LIN {X 0,Y 573.448,Z 568.908,A -85,B 0,C 180,E1 -2263.285,E2 -2263.285} C_VEL
LIN {X 0,Y 573.59,Z 558.034,A -85,B 0,C 180,E1 -2264.544,E2 -2264.544} C_VEL
LIN {X 0,Y 573.831,Z 547.069,A -85,B 0,C 180,E1 -2265.631,E2 -2265.631} C_VEL
LIN {X 0,Y 574.091,Z 533.22,A -85,B 0,C 180,E1 -2266.811,E2 -2266.811} C_VEL
LIN {X 0,Y 574.357,Z 519.267,A -85,B 0,C 180,E1 -2267.813,E2 -2267.813} C_VEL
LIN {X 0,Y 574.661,Z 505.713,A -85,B 0,C 180,E1 -2268.633,E2 -2268.633} C_VEL
LIN {X 0,Y 574.868,Z 491.148,A -85,B 0,C 180,E1 -2269.364,E2 -2269.364} C_VEL
LIN {X 0,Y 575.123,Z 475.242,A -85,B 0,C 180,E1 -2270.008,E2 -2270.008} C_VEL
LIN {X 0,Y 575.358,Z 459.013,A -85,B 0,C 180,E1 -2270.513,E2 -2270.513} C_VEL
LIN {X 0,Y 575.478,Z 442.433,A -85,B 0,C 180,E1 -2270.882,E2 -2270.882} C_VEL
LIN {X 0,Y 576.09,Z 283.124,A -85,B 0,C 180,E1 -2272.978,E2 -2272.978} C_VEL
LIN {X 0,Y 576.127,Z 240.798,A -85,B 0,C 180,E1 -2273.539,E2 -2273.539} C_VEL
LIN {X 0,Y 575.049,Z 234.756,A -85,B 0,C 180,E1 -2273.688,E2 -2273.688} C_VEL
LIN {X 0,Y 575.522,Z 200.414,A -85,B 0,C 180,E1 -2276.665,E2 -2276.665} C_VEL
LIN {X 0,Y 575.558,Z 194.845,A -85,B 0,C 180,E1 -2277.153,E2 -2277.153} C_VEL
LIN {X 0,Y 573.24,Z 186.394,A -85,B 0,C 180,E1 -2278.027,E2 -2278.027} C_VEL
LIN {X 0,Y 573.215,Z 186.397,A -85,B 0,C 180,E1 -2280.994,E2 -2280.994} C_VEL
LIN {X 0,Y 573.261,Z 186.39,A -85,B 0,C 180,E1 -2283.524,E2 -2283.524} C_VEL
LIN {X 0,Y 573.19,Z 186.394,A -85,B 0,C 180,E1 -2286.053,E2 -2286.053} C_VEL
LIN {X 0,Y 573.239,Z 186.391,A -85,B 0,C 180,E1 -2288.702,E2 -2288.702} C_VEL
LIN {X 0,Y 573.211,Z 186.393,A -85,B 0,C 180,E1 -2291.591,E2 -2291.591} C_VEL
LIN {X 0,Y 573.221,Z 186.39,A -85,B 0,C 180,E1 -2294.334,E2 -2294.334} C_VEL
LIN {X 0,Y 573.234,Z 186.392,A -85,B 0,C 180,E1 -2297.359,E2 -2297.359} C_VEL
LIN {X 0,Y 573.233,Z 186.389,A -85,B 0,C 180,E1 -2300.392,E2 -2300.392} C_VEL
LIN {X 0,Y 573.249,Z 186.391,A -85,B 0,C 180,E1 -2303.077,E2 -2303.077} C_VEL
LIN {X 0,Y 573.258,Z 186.385,A -85,B 0,C 180,E1 -2305.671,E2 -2305.671} C_VEL
LIN {X 0,Y 573.242,Z 186.386,A -85,B 0,C 180,E1 -2308.185,E2 -2308.185} C_VEL
LIN {X 0,Y 573.254,Z 186.392,A -85,B 0,C 180,E1 -2310.634,E2 -2310.634} C_VEL
LIN {X 0,Y 573.246,Z 186.388,A -85,B 0,C 180,E1 -2313.024,E2 -2313.024} C_VEL
LIN {X 0,Y 573.269,Z 186.383,A -85,B 0,C 180,E1 -2315.366,E2 -2315.366} C_VEL
LIN {X 0,Y 573.224,Z 186.395,A -85,B 0,C 180,E1 -2318.419,E2 -2318.419} C_VEL
LIN {X 0,Y 573.265,Z 186.389,A -85,B 0,C 180,E1 -2320.731,E2 -2320.731} C_VEL
LIN {X 0,Y 573.241,Z 186.386,A -85,B 0,C 180,E1 -2323.622,E2 -2323.622} C_VEL
LIN {X 0,Y 573.262,Z 186.385,A -85,B 0,C 180,E1 -2325.807,E2 -2325.807} C_VEL
LIN {X 0,Y 573.259,Z 186.387,A -85,B 0,C 180,E1 -2328.745,E2 -2328.745} C_VEL
LIN {X 0,Y 573.25,Z 186.385,A -85,B 0,C 180,E1 -2331.54,E2 -2331.54} C_VEL
LIN {X 0,Y 573.232,Z 186.388,A -85,B 0,C 180,E1 -2333.665,E2 -2333.665} C_VEL
LIN {X 0,Y 573.215,Z 186.389,A -85,B 0,C 180,E1 -2335.781,E2 -2335.781} C_VEL
LIN {X 0,Y 573.297,Z 186.377,A -85,B 0,C 180,E1 -2337.892,E2 -2337.892} C_VEL
LIN {X 0,Y 573.332,Z 186.378,A -85,B 0,C 180,E1 -2340.702,E2 -2340.702} C_VEL
LIN {X 0,Y 573.226,Z 186.389,A -85,B 0,C 180,E1 -2343.515,E2 -2343.515} C_VEL
LIN {X 0,Y 573.282,Z 186.38,A -85,B 0,C 180,E1 -2345.628,E2 -2345.628} C_VEL
LIN {X 0,Y 573.28,Z 186.386,A -85,B 0,C 180,E1 -2348.46,E2 -2348.46} C_VEL
LIN {X 0,Y 573.268,Z 186.382,A -85,B 0,C 180,E1 -2351.312,E2 -2351.312} C_VEL
LIN {X 0,Y 573.278,Z 186.386,A -85,B 0,C 180,E1 -2354.424,E2 -2354.424} C_VEL
LIN {X 0,Y 573.256,Z 186.384,A -85,B 0,C 180,E1 -2357.112,E2 -2357.112} C_VEL
LIN {X 0,Y 573.249,Z 186.393,A -85,B 0,C 180,E1 -2360.077,E2 -2360.077} C_VEL
LIN {X 0,Y 573.231,Z 186.388,A -85,B 0,C 180,E1 -2363.099,E2 -2363.099} C_VEL
LIN {X 0,Y 573.248,Z 186.386,A -85,B 0,C 180,E1 -2364.392,E2 -2364.392} C_VEL
LIN {X 0,Y 572.62,Z 186.463,A -85,B 0,C 180,E1 -2364.979,E2 -2364.979} C_VEL
LIN {X 0,Y 569.777,Z 186.825,A -85,B 0,C 180,E1 -2365.93,E2 -2365.93} C_VEL
LIN {X 0,Y 567.347,Z 187.126,A -85,B 0,C 180,E1 -2366.696,E2 -2366.696} C_VEL
LIN {X 0,Y 566.297,Z 187.253,A -85,B 0,C 180,E1 -2367.287,E2 -2367.287} C_VEL
LIN {X 0,Y 566.209,Z 187.264,A -85,B 0,C 180,E1 -2367.487,E2 -2367.487} C_VEL
LIN {X 0,Y 566.223,Z 187.27,A -85,B 0,C 180,E1 -2369.767,E2 -2369.767} C_VEL
LIN {X 0,Y 566.202,Z 187.262,A -85,B 0,C 180,E1 -2372.43,E2 -2372.43} C_VEL
LIN {X 0,Y 566.21,Z 187.263,A -85,B 0,C 180,E1 -2374.994,E2 -2374.994} C_VEL
LIN {X 0,Y 566.194,Z 187.271,A -85,B 0,C 180,E1 -2377.461,E2 -2377.461} C_VEL
LIN {X 0,Y 566.204,Z 187.265,A -85,B 0,C 180,E1 -2380.199,E2 -2380.199} C_VEL
LIN {X 0,Y 566.197,Z 187.266,A -85,B 0,C 180,E1 -2383.054,E2 -2383.054} C_VEL
LIN {X 0,Y 566.196,Z 187.267,A -85,B 0,C 180,E1 -2386.049,E2 -2386.049} C_VEL
LIN {X 0,Y 566.202,Z 187.268,A -85,B 0,C 180,E1 -2389.215,E2 -2389.215} C_VEL
LIN {X 0,Y 566.184,Z 187.272,A -85,B 0,C 180,E1 -2391.637,E2 -2391.637} C_VEL
LIN {X 0,Y 566.164,Z 187.267,A -85,B 0,C 180,E1 -2394.308,E2 -2394.308} C_VEL
LIN {X 0,Y 566.227,Z 187.264,A -85,B 0,C 180,E1 -2396.899,E2 -2396.899} C_VEL
LIN {X 0,Y 566.183,Z 187.274,A -85,B 0,C 180,E1 -2399.408,E2 -2399.408} C_VEL
LIN {X 0,Y 566.21,Z 187.263,A -85,B 0,C 180,E1 -2401.857,E2 -2401.857} C_VEL
LIN {X 0,Y 566.215,Z 187.262,A -85,B 0,C 180,E1 -2404.251,E2 -2404.251} C_VEL
LIN {X 0,Y 566.173,Z 187.269,A -85,B 0,C 180,E1 -2406.718,E2 -2406.718} C_VEL
LIN {X 0,Y 566.206,Z 187.262,A -85,B 0,C 180,E1 -2409.663,E2 -2409.663} C_VEL
LIN {X 0,Y 566.198,Z 187.267,A -85,B 0,C 180,E1 -2412.668,E2 -2412.668} C_VEL
LIN {X 0,Y 566.234,Z 187.257,A -85,B 0,C 180,E1 -2415.627,E2 -2415.627} C_VEL
LIN {X 0,Y 566.235,Z 187.266,A -85,B 0,C 180,E1 -2418.675,E2 -2418.675} C_VEL
LIN {X 0,Y 566.227,Z 187.264,A -85,B 0,C 180,E1 -2421.434,E2 -2421.434} C_VEL
LIN {X 0,Y 566.264,Z 187.257,A -85,B 0,C 180,E1 -2424.302,E2 -2424.302} C_VEL
LIN {X 0,Y 566.283,Z 187.256,A -85,B 0,C 180,E1 -2427.866,E2 -2427.866} C_VEL
LIN {X 0,Y 566.29,Z 187.349,A -85,B 0,C 180,E1 -2430.111,E2 -2430.111} C_VEL
LIN {X 0,Y 568.261,Z 195.71,A -85,B 0,C 180,E1 -2431.063,E2 -2431.063} C_VEL
LIN {X 0,Y 568.073,Z 205.902,A -85,B 0,C 180,E1 -2432.082,E2 -2432.082} C_VEL
LIN {X 0,Y 569.715,Z 214.515,A -85,B 0,C 180,E1 -2432.275,E2 -2432.275} C_VEL
LIN {X 0,Y 568.912,Z 411.289,A -85,B 0,C 180,E1 -2434.894,E2 -2434.894} C_VEL
LIN {X 0,Y 568.729,Z 427.818,A -85,B 0,C 180,E1 -2435.251,E2 -2435.251} C_VEL
LIN {X 0,Y 568.454,Z 443.359,A -85,B 0,C 180,E1 -2435.72,E2 -2435.72} C_VEL
LIN {X 0,Y 568.214,Z 459.109,A -85,B 0,C 180,E1 -2436.346,E2 -2436.346} C_VEL
LIN {X 0,Y 567.874,Z 474.384,A -85,B 0,C 180,E1 -2437.109,E2 -2437.109} C_VEL
LIN {X 0,Y 567.574,Z 488.661,A -85,B 0,C 180,E1 -2437.973,E2 -2437.973} C_VEL
LIN {X 0,Y 567.234,Z 502.895,A -85,B 0,C 180,E1 -2438.999,E2 -2438.999} C_VEL
LIN {X 0,Y 566.989,Z 514.689,A -85,B 0,C 180,E1 -2439.993,E2 -2439.993} C_VEL
LIN {X 0,Y 566.695,Z 527.464,A -85,B 0,C 180,E1 -2441.258,E2 -2441.258} C_VEL
LIN {X 0,Y 566.452,Z 538.47,A -85,B 0,C 180,E1 -2442.54,E2 -2442.54} C_VEL
LIN {X 0,Y 566.289,Z 547.928,A -85,B 0,C 180,E1 -2443.821,E2 -2443.821} C_VEL
LIN {X 0,Y 566.129,Z 557.174,A -85,B 0,C 180,E1 -2445.295,E2 -2445.295} C_VEL
LIN {X 0,Y 566.032,Z 565.16,A -85,B 0,C 180,E1 -2446.82,E2 -2446.82} C_VEL
LIN {X 0,Y 565.958,Z 572.1,A -85,B 0,C 180,E1 -2448.46,E2 -2448.46} C_VEL
LIN {X 0,Y 565.918,Z 577.139,A -85,B 0,C 180,E1 -2449.969,E2 -2449.969} C_VEL
LIN {X 0,Y 565.861,Z 580.733,A -85,B 0,C 180,E1 -2451.331,E2 -2451.331} C_VEL
LIN {X 0,Y 565.827,Z 584.092,A -85,B 0,C 180,E1 -2453.201,E2 -2453.201} C_VEL
LIN {X 0,Y 565.809,Z 585.689,A -85,B 0,C 180,E1 -2454.941,E2 -2454.941} C_VEL
LIN {X 0,Y 565.854,Z 585.887,A -85,B 0,C 180,E1 -2456.588,E2 -2456.588} C_VEL
LIN {X 0,Y 565.826,Z 584.912,A -85,B 0,C 180,E1 -2458.163,E2 -2458.163} C_VEL
LIN {X 0,Y 565.866,Z 582.694,A -85,B 0,C 180,E1 -2459.788,E2 -2459.788} C_VEL
LIN {X 0,Y 565.93,Z 579.049,A -85,B 0,C 180,E1 -2461.437,E2 -2461.437} C_VEL
LIN {X 0,Y 565.903,Z 573.917,A -85,B 0,C 180,E1 -2463.122,E2 -2463.122} C_VEL
LIN {X 0,Y 565.974,Z 569.043,A -85,B 0,C 180,E1 -2464.401,E2 -2464.401} C_VEL
LIN {X 0,Y 566.052,Z 561.787,A -85,B 0,C 180,E1 -2465.947,E2 -2465.947} C_VEL
LIN {X 0,Y 566.173,Z 553.186,A -85,B 0,C 180,E1 -2467.462,E2 -2467.462} C_VEL
LIN {X 0,Y 566.333,Z 543.574,A -85,B 0,C 180,E1 -2468.883,E2 -2468.883} C_VEL
LIN {X 0,Y 566.572,Z 532.373,A -85,B 0,C 180,E1 -2470.283,E2 -2470.283} C_VEL
LIN {X 0,Y 566.812,Z 520.413,A -85,B 0,C 180,E1 -2471.555,E2 -2471.555} C_VEL
LIN {X 0,Y 567.142,Z 507.509,A -85,B 0,C 180,E1 -2472.722,E2 -2472.722} C_VEL
LIN {X 0,Y 567.435,Z 493.68,A -85,B 0,C 180,E1 -2473.779,E2 -2473.779} C_VEL
LIN {X 0,Y 567.751,Z 480.14,A -85,B 0,C 180,E1 -2474.651,E2 -2474.651} C_VEL
LIN {X 0,Y 568.074,Z 464.55,A -85,B 0,C 180,E1 -2475.488,E2 -2475.488} C_VEL
LIN {X 0,Y 568.38,Z 448.583,A -85,B 0,C 180,E1 -2476.177,E2 -2476.177} C_VEL
LIN {X 0,Y 568.643,Z 432.346,A -85,B 0,C 180,E1 -2476.72,E2 -2476.72} C_VEL
LIN {X 0,Y 568.874,Z 415.406,A -85,B 0,C 180,E1 -2477.124,E2 -2477.124} C_VEL
LIN {X 0,Y 568.979,Z 392.613,A -85,B 0,C 180,E1 -2477.462,E2 -2477.462} C_VEL
LIN {X 0,Y 569.624,Z 213.633,A -85,B 0,C 180,E1 -2479.831,E2 -2479.831} C_VEL
LIN {X 0,Y 568.055,Z 205.768,A -85,B 0,C 180,E1 -2480.023,E2 -2480.023} C_VEL
LIN {X 0,Y 568.193,Z 195.363,A -85,B 0,C 180,E1 -2481.069,E2 -2481.069} C_VEL
LIN {X 0,Y 566.192,Z 187.271,A -85,B 0,C 180,E1 -2482.005,E2 -2482.005} C_VEL
LIN {X 0,Y 566.188,Z 187.274,A -85,B 0,C 180,E1 -2485.181,E2 -2485.181} C_VEL
LIN {X 0,Y 566.219,Z 187.265,A -85,B 0,C 180,E1 -2487.743,E2 -2487.743} C_VEL
LIN {X 0,Y 566.163,Z 187.271,A -85,B 0,C 180,E1 -2490.333,E2 -2490.333} C_VEL
LIN {X 0,Y 566.162,Z 187.274,A -85,B 0,C 180,E1 -2492.658,E2 -2492.658} C_VEL
LIN {X 0,Y 566.185,Z 187.274,A -85,B 0,C 180,E1 -2495.037,E2 -2495.037} C_VEL
LIN {X 0,Y 566.179,Z 187.266,A -85,B 0,C 180,E1 -2498.137,E2 -2498.137} C_VEL
LIN {X 0,Y 566.222,Z 187.269,A -85,B 0,C 180,E1 -2500.614,E2 -2500.614} C_VEL
LIN {X 0,Y 566.203,Z 187.264,A -85,B 0,C 180,E1 -2503.412,E2 -2503.412} C_VEL
LIN {X 0,Y 566.184,Z 187.271,A -85,B 0,C 180,E1 -2506.359,E2 -2506.359} C_VEL
LIN {X 0,Y 566.227,Z 187.268,A -85,B 0,C 180,E1 -2508.675,E2 -2508.675} C_VEL
LIN {X 0,Y 566.197,Z 187.264,A -85,B 0,C 180,E1 -2511.434,E2 -2511.434} C_VEL
LIN {X 0,Y 566.249,Z 187.265,A -85,B 0,C 180,E1 -2514.302,E2 -2514.302} C_VEL
LIN {X 0,Y 566.267,Z 187.258,A -85,B 0,C 180,E1 -2517.866,E2 -2517.866} C_VEL
LIN {X 0,Y 566.3,Z 187.255,A -85,B 0,C 180,E1 -2520.711,E2 -2520.711} C_VEL
LIN {X 0,Y 566.269,Z 187.256,A -85,B 0,C 180,E1 -2522.846,E2 -2522.846} C_VEL
LIN {X 0,Y 566.249,Z 187.261,A -85,B 0,C 180,E1 -2525.698,E2 -2525.698} C_VEL
LIN {X 0,Y 566.227,Z 187.263,A -85,B 0,C 180,E1 -2528.566,E2 -2528.566} C_VEL
LIN {X 0,Y 566.235,Z 187.261,A -85,B 0,C 180,E1 -2531.454,E2 -2531.454} C_VEL
LIN {X 0,Y 566.228,Z 187.263,A -85,B 0,C 180,E1 -2534.507,E2 -2534.507} C_VEL
LIN {X 0,Y 566.197,Z 187.266,A -85,B 0,C 180,E1 -2537.332,E2 -2537.332} C_VEL
LIN {X 0,Y 566.207,Z 187.265,A -85,B 0,C 180,E1 -2540.337,E2 -2540.337} C_VEL
LIN {X 0,Y 566.183,Z 187.271,A -85,B 0,C 180,E1 -2543.404,E2 -2543.404} C_VEL
LIN {X 0,Y 566.22,Z 187.269,A -85,B 0,C 180,E1 -2545.749,E2 -2545.749} C_VEL
LIN {X 0,Y 566.2,Z 187.266,A -85,B 0,C 180,E1 -2548.203,E2 -2548.203} C_VEL
LIN {X 0,Y 566.193,Z 187.269,A -85,B 0,C 180,E1 -2551.078,E2 -2551.078} C_VEL
LIN {X 0,Y 566.215,Z 187.265,A -85,B 0,C 180,E1 -2553.955,E2 -2553.955} C_VEL
LIN {X 0,Y 566.194,Z 187.266,A -85,B 0,C 180,E1 -2556.57,E2 -2556.57} C_VEL
LIN {X 0,Y 566.215,Z 187.273,A -85,B 0,C 180,E1 -2559.273,E2 -2559.273} C_VEL
LIN {X 0,Y 566.184,Z 187.268,A -85,B 0,C 180,E1 -2562.09,E2 -2562.09} C_VEL
LIN {X 0,Y 566.167,Z 187.278,A -85,B 0,C 180,E1 -2565.036,E2 -2565.036} C_VEL
LIN {X 0,Y 566.184,Z 187.268,A -85,B 0,C 180,E1 -2567.911,E2 -2567.911} C_VEL
LIN {X 0,Y 566.215,Z 187.269,A -85,B 0,C 180,E1 -2570.727,E2 -2570.727} C_VEL
LIN {X 0,Y 566.179,Z 187.268,A -85,B 0,C 180,E1 -2573.789,E2 -2573.789} C_VEL
LIN {X 0,Y 566.207,Z 187.265,A -85,B 0,C 180,E1 -2576.266,E2 -2576.266} C_VEL
LIN {X 0,Y 566.187,Z 187.275,A -85,B 0,C 180,E1 -2578.924,E2 -2578.924} C_VEL
LIN {X 0,Y 566.209,Z 187.455,A -85,B 0,C 180,E1 -2581.722,E2 -2581.722} C_VEL
LIN {X 0,Y 568.721,Z 195.965,A -85,B 0,C 180,E1 -2582.613,E2 -2582.613} C_VEL
LIN {X 0,Y 568.851,Z 202.776,A -85,B 0,C 180,E1 -2583.226,E2 -2583.226} C_VEL
LIN {X 0,Y 568.332,Z 234.996,A -85,B 0,C 180,E1 -2586.036,E2 -2586.036} C_VEL
LIN {X 0,Y 569.708,Z 242.837,A -85,B 0,C 180,E1 -2586.207,E2 -2586.207} C_VEL
LIN {X 0,Y 568.89,Z 442.456,A -85,B 0,C 180,E1 -2588.865,E2 -2588.865} C_VEL
LIN {X 0,Y 568.721,Z 459.026,A -85,B 0,C 180,E1 -2589.237,E2 -2589.237} C_VEL
LIN {X 0,Y 568.422,Z 475.253,A -85,B 0,C 180,E1 -2589.746,E2 -2589.746} C_VEL
LIN {X 0,Y 568.144,Z 491.394,A -85,B 0,C 180,E1 -2590.409,E2 -2590.409} C_VEL
LIN {X 0,Y 567.877,Z 505.721,A -85,B 0,C 180,E1 -2591.137,E2 -2591.137} C_VEL
LIN {X 0,Y 567.582,Z 519.277,A -85,B 0,C 180,E1 -2591.968,E2 -2591.968} C_VEL
LIN {X 0,Y 567.227,Z 533.222,A -85,B 0,C 180,E1 -2592.98,E2 -2592.98} C_VEL
LIN {X 0,Y 566.915,Z 547.073,A -85,B 0,C 180,E1 -2594.174,E2 -2594.174} C_VEL
LIN {X 0,Y 566.63,Z 558.622,A -85,B 0,C 180,E1 -2595.34,E2 -2595.34} C_VEL
LIN {X 0,Y 566.434,Z 570.34,A -85,B 0,C 180,E1 -2596.731,E2 -2596.731} C_VEL
LIN {X 0,Y 566.238,Z 580.674,A -85,B 0,C 180,E1 -2598.183,E2 -2598.183} C_VEL
LIN {X 0,Y 566.119,Z 589.286,A -85,B 0,C 180,E1 -2599.63,E2 -2599.63} C_VEL
LIN {X 0,Y 566.001,Z 596.491,A -85,B 0,C 180,E1 -2601.071,E2 -2601.071} C_VEL
LIN {X 0,Y 565.967,Z 602.467,A -85,B 0,C 180,E1 -2602.508,E2 -2602.508} C_VEL
LIN {X 0,Y 565.916,Z 607.188,A -85,B 0,C 180,E1 -2603.941,E2 -2603.941} C_VEL
LIN {X 0,Y 565.91,Z 611.637,A -85,B 0,C 180,E1 -2605.727,E2 -2605.727} C_VEL
LIN {X 0,Y 565.865,Z 614.09,A -85,B 0,C 180,E1 -2607.153,E2 -2607.153} C_VEL
LIN {X 0,Y 565.839,Z 615.48,A -85,B 0,C 180,E1 -2608.577,E2 -2608.577} C_VEL
LIN {X 0,Y 565.834,Z 616,A -85,B 0,C 180,E1 -2610,E2 -2610} C_VEL
LIN {X 0,Y 565.839,Z 615.48,A -85,B 0,C 180,E1 -2611.424,E2 -2611.424} C_VEL
LIN {X 0,Y 565.866,Z 614.088,A -85,B 0,C 180,E1 -2612.848,E2 -2612.848} C_VEL
LIN {X 0,Y 565.91,Z 611.636,A -85,B 0,C 180,E1 -2614.273,E2 -2614.273} C_VEL
LIN {X 0,Y 565.915,Z 607.188,A -85,B 0,C 180,E1 -2616.06,E2 -2616.06} C_VEL
LIN {X 0,Y 565.968,Z 602.467,A -85,B 0,C 180,E1 -2617.492,E2 -2617.492} C_VEL
LIN {X 0,Y 566.002,Z 596.489,A -85,B 0,C 180,E1 -2618.929,E2 -2618.929} C_VEL
LIN {X 0,Y 566.126,Z 588.276,A -85,B 0,C 180,E1 -2620.551,E2 -2620.551} C_VEL
LIN {X 0,Y 566.246,Z 579.442,A -85,B 0,C 180,E1 -2621.999,E2 -2621.999} C_VEL
LIN {X 0,Y 566.427,Z 568.907,A -85,B 0,C 180,E1 -2623.453,E2 -2623.453} C_VEL
LIN {X 0,Y 566.661,Z 557.611,A -85,B 0,C 180,E1 -2624.774,E2 -2624.774} C_VEL
LIN {X 0,Y 566.958,Z 545.117,A -85,B 0,C 180,E1 -2626.01,E2 -2626.01} C_VEL
LIN {X 0,Y 567.229,Z 532.044,A -85,B 0,C 180,E1 -2627.113,E2 -2627.113} C_VEL
LIN {X 0,Y 567.585,Z 517.849,A -85,B 0,C 180,E1 -2628.126,E2 -2628.126} C_VEL
LIN {X 0,Y 567.9,Z 504.028,A -85,B 0,C 180,E1 -2628.957,E2 -2628.957} C_VEL
LIN {X 0,Y 568.197,Z 489.524,A -85,B 0,C 180,E1 -2629.678,E2 -2629.678} C_VEL
LIN {X 0,Y 568.462,Z 473.942,A -85,B 0,C 180,E1 -2630.3,E2 -2630.3} C_VEL
LIN {X 0,Y 568.724,Z 457.183,A -85,B 0,C 180,E1 -2630.81,E2 -2630.81} C_VEL
LIN {X 0,Y 568.855,Z 440.942,A -85,B 0,C 180,E1 -2631.161,E2 -2631.161} C_VEL
LIN {X 0,Y 569.681,Z 242.973,A -85,B 0,C 180,E1 -2633.793,E2 -2633.793} C_VEL
LIN {X 0,Y 568.343,Z 234.838,A -85,B 0,C 180,E1 -2633.978,E2 -2633.978} C_VEL
LIN {X 0,Y 568.91,Z 199.819,A -85,B 0,C 180,E1 -2637.037,E2 -2637.037} C_VEL
LIN {X 0,Y 568.937,Z 197.003,A -85,B 0,C 180,E1 -2637.287,E2 -2637.287} C_VEL
LIN {X 0,Y 566.202,Z 187.271,A -85,B 0,C 180,E1 -2638.324,E2 -2638.324} C_VEL
LIN {X 0,Y 566.185,Z 187.272,A -85,B 0,C 180,E1 -2641.422,E2 -2641.422} C_VEL
LIN {X 0,Y 566.204,Z 187.265,A -85,B 0,C 180,E1 -2643.956,E2 -2643.956} C_VEL
LIN {X 0,Y 566.179,Z 187.27,A -85,B 0,C 180,E1 -2646.571,E2 -2646.571} C_VEL
LIN {X 0,Y 566.214,Z 187.263,A -85,B 0,C 180,E1 -2649.686,E2 -2649.686} C_VEL
LIN {X 0,Y 566.189,Z 187.272,A -85,B 0,C 180,E1 -2652.916,E2 -2652.916} C_VEL
LIN {X 0,Y 566.158,Z 187.268,A -85,B 0,C 180,E1 -2655.961,E2 -2655.961} C_VEL
LIN {X 0,Y 566.182,Z 187.267,A -85,B 0,C 180,E1 -2658.14,E2 -2658.14} C_VEL
LIN {X 0,Y 566.208,Z 187.268,A -85,B 0,C 180,E1 -2660.726,E2 -2660.726} C_VEL
LIN {X 0,Y 566.18,Z 187.264,A -85,B 0,C 180,E1 -2663.788,E2 -2663.788} C_VEL
LIN {X 0,Y 566.194,Z 187.267,A -85,B 0,C 180,E1 -2666.268,E2 -2666.268} C_VEL
LIN {X 0,Y 566.189,Z 187.272,A -85,B 0,C 180,E1 -2668.923,E2 -2668.923} C_VEL
LIN {X 0,Y 566.208,Z 187.263,A -85,B 0,C 180,E1 -2671.857,E2 -2671.857} C_VEL
LIN {X 0,Y 566.204,Z 187.263,A -85,B 0,C 180,E1 -2674.251,E2 -2674.251} C_VEL
LIN {X 0,Y 566.168,Z 187.277,A -85,B 0,C 180,E1 -2676.719,E2 -2676.719} C_VEL
LIN {X 0,Y 566.202,Z 187.261,A -85,B 0,C 180,E1 -2679.663,E2 -2679.663} C_VEL
LIN {X 0,Y 566.195,Z 187.273,A -85,B 0,C 180,E1 -2682.668,E2 -2682.668} C_VEL
LIN {X 0,Y 566.224,Z 187.26,A -85,B 0,C 180,E1 -2685.627,E2 -2685.627} C_VEL
LIN {X 0,Y 566.231,Z 187.263,A -85,B 0,C 180,E1 -2688.675,E2 -2688.675} C_VEL
LIN {X 0,Y 566.201,Z 187.263,A -85,B 0,C 180,E1 -2691.434,E2 -2691.434} C_VEL
LIN {X 0,Y 566.252,Z 187.266,A -85,B 0,C 180,E1 -2694.302,E2 -2694.302} C_VEL
LIN {X 0,Y 566.269,Z 187.252,A -85,B 0,C 180,E1 -2697.866,E2 -2697.866} C_VEL
LIN {X 0,Y 566.302,Z 187.254,A -85,B 0,C 180,E1 -2700.711,E2 -2700.711} C_VEL
LIN {X 0,Y 566.27,Z 187.256,A -85,B 0,C 180,E1 -2702.846,E2 -2702.846} C_VEL
LIN {X 0,Y 566.251,Z 187.256,A -85,B 0,C 180,E1 -2705.698,E2 -2705.698} C_VEL
LIN {X 0,Y 566.224,Z 187.264,A -85,B 0,C 180,E1 -2708.566,E2 -2708.566} C_VEL
LIN {X 0,Y 566.239,Z 187.258,A -85,B 0,C 180,E1 -2711.454,E2 -2711.454} C_VEL
LIN {X 0,Y 566.231,Z 187.262,A -85,B 0,C 180,E1 -2714.507,E2 -2714.507} C_VEL
LIN {X 0,Y 566.2,Z 187.264,A -85,B 0,C 180,E1 -2717.332,E2 -2717.332} C_VEL
LIN {X 0,Y 566.21,Z 187.265,A -85,B 0,C 180,E1 -2720.337,E2 -2720.337} C_VEL
LIN {X 0,Y 566.187,Z 187.268,A -85,B 0,C 180,E1 -2723.404,E2 -2723.404} C_VEL
LIN {X 0,Y 566.212,Z 187.268,A -85,B 0,C 180,E1 -2725.749,E2 -2725.749} C_VEL
LIN {X 0,Y 566.209,Z 187.264,A -85,B 0,C 180,E1 -2727.487,E2 -2727.487} C_VEL
LIN {X 0,Y 565.534,Z 187.353,A -85,B 0,C 180,E1 -2728.081,E2 -2728.081} C_VEL
LIN {X 0,Y 562.671,Z 187.704,A -85,B 0,C 180,E1 -2729.045,E2 -2729.045} C_VEL
LIN {X 0,Y 560.258,Z 188.012,A -85,B 0,C 180,E1 -2729.82,E2 -2729.82} C_VEL
LIN {X 0,Y 559.226,Z 188.133,A -85,B 0,C 180,E1 -2730.419,E2 -2730.419} C_VEL
LIN {X 0,Y 559.144,Z 188.142,A -85,B 0,C 180,E1 -2730.622,E2 -2730.622} C_VEL
LIN {X 0,Y 559.162,Z 188.146,A -85,B 0,C 180,E1 -2733.575,E2 -2733.575} C_VEL
LIN {X 0,Y 559.166,Z 188.14,A -85,B 0,C 180,E1 -2736.449,E2 -2736.449} C_VEL
LIN {X 0,Y 559.171,Z 188.138,A -85,B 0,C 180,E1 -2738.934,E2 -2738.934} C_VEL
LIN {X 0,Y 559.174,Z 188.14,A -85,B 0,C 180,E1 -2742.137,E2 -2742.137} C_VEL
LIN {X 0,Y 559.136,Z 188.148,A -85,B 0,C 180,E1 -2745.261,E2 -2745.261} C_VEL
LIN {X 0,Y 559.164,Z 188.139,A -85,B 0,C 180,E1 -2748.23,E2 -2748.23} C_VEL
LIN {X 0,Y 559.172,Z 188.145,A -85,B 0,C 180,E1 -2751.192,E2 -2751.192} C_VEL
LIN {X 0,Y 559.138,Z 188.145,A -85,B 0,C 180,E1 -2753.789,E2 -2753.789} C_VEL
LIN {X 0,Y 559.164,Z 188.141,A -85,B 0,C 180,E1 -2756.425,E2 -2756.425} C_VEL
LIN {X 0,Y 559.157,Z 188.144,A -85,B 0,C 180,E1 -2758.981,E2 -2758.981} C_VEL
LIN {X 0,Y 559.167,Z 188.143,A -85,B 0,C 180,E1 -2761.619,E2 -2761.619} C_VEL
LIN {X 0,Y 559.182,Z 188.139,A -85,B 0,C 180,E1 -2763.903,E2 -2763.903} C_VEL
LIN {X 0,Y 559.142,Z 188.143,A -85,B 0,C 180,E1 -2766.571,E2 -2766.571} C_VEL
LIN {X 0,Y 559.175,Z 188.141,A -85,B 0,C 180,E1 -2769.395,E2 -2769.395} C_VEL
LIN {X 0,Y 559.141,Z 188.143,A -85,B 0,C 180,E1 -2771.686,E2 -2771.686} C_VEL
LIN {X 0,Y 559.161,Z 188.142,A -85,B 0,C 180,E1 -2773.948,E2 -2773.948} C_VEL
LIN {X 0,Y 559.172,Z 188.135,A -85,B 0,C 180,E1 -2776.184,E2 -2776.184} C_VEL
LIN {X 0,Y 559.194,Z 188.144,A -85,B 0,C 180,E1 -2779.133,E2 -2779.133} C_VEL
LIN {X 0,Y 559.204,Z 188.137,A -85,B 0,C 180,E1 -2782.054,E2 -2782.054} C_VEL
LIN {X 0,Y 559.251,Z 188.138,A -85,B 0,C 180,E1 -2784.953,E2 -2784.953} C_VEL
LIN {X 0,Y 559.254,Z 188.132,A -85,B 0,C 180,E1 -2787.839,E2 -2787.839} C_VEL
LIN {X 0,Y 559.277,Z 188.293,A -85,B 0,C 180,E1 -2789.842,E2 -2789.842} C_VEL
LIN {X 0,Y 561.531,Z 197.362,A -85,B 0,C 180,E1 -2790.896,E2 -2790.896} C_VEL
LIN {X 0,Y 561.404,Z 205.971,A -85,B 0,C 180,E1 -2791.77,E2 -2791.77} C_VEL
LIN {X 0,Y 563.214,Z 215.618,A -85,B 0,C 180,E1 -2791.997,E2 -2791.997} C_VEL
LIN {X 0,Y 562.284,Z 410.249,A -85,B 0,C 180,E1 -2794.615,E2 -2794.615} C_VEL
LIN {X 0,Y 562.114,Z 426.297,A -85,B 0,C 180,E1 -2794.953,E2 -2794.953} C_VEL
LIN {X 0,Y 561.806,Z 442.267,A -85,B 0,C 180,E1 -2795.428,E2 -2795.428} C_VEL
LIN {X 0,Y 561.504,Z 458.202,A -85,B 0,C 180,E1 -2796.062,E2 -2796.062} C_VEL
LIN {X 0,Y 561.127,Z 473.669,A -85,B 0,C 180,E1 -2796.833,E2 -2796.833} C_VEL
LIN {X 0,Y 560.794,Z 487.9,A -85,B 0,C 180,E1 -2797.696,E2 -2797.696} C_VEL
LIN {X 0,Y 560.449,Z 501.272,A -85,B 0,C 180,E1 -2798.654,E2 -2798.654} C_VEL
LIN {X 0,Y 560.093,Z 514.278,A -85,B 0,C 180,E1 -2799.752,E2 -2799.752} C_VEL
LIN {X 0,Y 559.742,Z 526.979,A -85,B 0,C 180,E1 -2801.019,E2 -2801.019} C_VEL
LIN {X 0,Y 559.482,Z 538.164,A -85,B 0,C 180,E1 -2802.33,E2 -2802.33} C_VEL
LIN {X 0,Y 559.257,Z 548.906,A -85,B 0,C 180,E1 -2803.813,E2 -2803.813} C_VEL
LIN {X 0,Y 559.064,Z 557.999,A -85,B 0,C 180,E1 -2805.307,E2 -2805.307} C_VEL
LIN {X 0,Y 558.954,Z 565.642,A -85,B 0,C 180,E1 -2806.809,E2 -2806.809} C_VEL
LIN {X 0,Y 558.871,Z 571.942,A -85,B 0,C 180,E1 -2808.323,E2 -2808.323} C_VEL
LIN {X 0,Y 558.84,Z 577.015,A -85,B 0,C 180,E1 -2809.849,E2 -2809.849} C_VEL
LIN {X 0,Y 558.766,Z 581.099,A -85,B 0,C 180,E1 -2811.448,E2 -2811.448} C_VEL
LIN {X 0,Y 558.728,Z 583.766,A -85,B 0,C 180,E1 -2812.95,E2 -2812.95} C_VEL
LIN {X 0,Y 558.697,Z 585.428,A -85,B 0,C 180,E1 -2814.526,E2 -2814.526} C_VEL
LIN {X 0,Y 558.73,Z 585.99,A -85,B 0,C 180,E1 -2816.119,E2 -2816.119} C_VEL
LIN {X 0,Y 558.728,Z 585.315,A -85,B 0,C 180,E1 -2817.736,E2 -2817.736} C_VEL
LIN {X 0,Y 558.759,Z 583.406,A -85,B 0,C 180,E1 -2819.375,E2 -2819.375} C_VEL
LIN {X 0,Y 558.788,Z 580.19,A -85,B 0,C 180,E1 -2821.041,E2 -2821.041} C_VEL
LIN {X 0,Y 558.806,Z 575.529,A -85,B 0,C 180,E1 -2822.738,E2 -2822.738} C_VEL
LIN {X 0,Y 558.897,Z 570.434,A -85,B 0,C 180,E1 -2824.155,E2 -2824.155} C_VEL
LIN {X 0,Y 558.978,Z 563.254,A -85,B 0,C 180,E1 -2825.777,E2 -2825.777} C_VEL
LIN {X 0,Y 559.097,Z 554.569,A -85,B 0,C 180,E1 -2827.378,E2 -2827.378} C_VEL
LIN {X 0,Y 559.301,Z 545.183,A -85,B 0,C 180,E1 -2828.824,E2 -2828.824} C_VEL
LIN {X 0,Y 559.524,Z 535.207,A -85,B 0,C 180,E1 -2830.131,E2 -2830.131} C_VEL
LIN {X 0,Y 559.795,Z 524.126,A -85,B 0,C 180,E1 -2831.372,E2 -2831.372} C_VEL
LIN {X 0,Y 560.126,Z 512.299,A -85,B 0,C 180,E1 -2832.513,E2 -2832.513} C_VEL
LIN {X 0,Y 560.474,Z 499.121,A -85,B 0,C 180,E1 -2833.603,E2 -2833.603} C_VEL
LIN {X 0,Y 560.833,Z 485.319,A -85,B 0,C 180,E1 -2834.567,E2 -2834.567} C_VEL
LIN {X 0,Y 561.168,Z 471.555,A -85,B 0,C 180,E1 -2835.372,E2 -2835.372} C_VEL
LIN {X 0,Y 561.566,Z 455.341,A -85,B 0,C 180,E1 -2836.151,E2 -2836.151} C_VEL
LIN {X 0,Y 561.875,Z 438.977,A -85,B 0,C 180,E1 -2836.768,E2 -2836.768} C_VEL
LIN {X 0,Y 562.127,Z 423.201,A -85,B 0,C 180,E1 -2837.216,E2 -2837.216} C_VEL
LIN {X 0,Y 562.339,Z 406.167,A -85,B 0,C 180,E1 -2837.543,E2 -2837.543} C_VEL
LIN {X 0,Y 563.174,Z 215.452,A -85,B 0,C 180,E1 -2840.097,E2 -2840.097} C_VEL
LIN {X 0,Y 561.373,Z 206.023,A -85,B 0,C 180,E1 -2840.321,E2 -2840.321} C_VEL
LIN {X 0,Y 561.408,Z 196.947,A -85,B 0,C 180,E1 -2841.25,E2 -2841.25} C_VEL
LIN {X 0,Y 559.14,Z 188.149,A -85,B 0,C 180,E1 -2842.311,E2 -2842.311} C_VEL
LIN {X 0,Y 559.128,Z 188.15,A -85,B 0,C 180,E1 -2845.554,E2 -2845.554} C_VEL
LIN {X 0,Y 559.154,Z 188.144,A -85,B 0,C 180,E1 -2848.137,E2 -2848.137} C_VEL
LIN {X 0,Y 559.11,Z 188.152,A -85,B 0,C 180,E1 -2850.644,E2 -2850.644} C_VEL
LIN {X 0,Y 559.116,Z 188.154,A -85,B 0,C 180,E1 -2853.182,E2 -2853.182} C_VEL
LIN {X 0,Y 559.113,Z 188.15,A -85,B 0,C 180,E1 -2855.493,E2 -2855.493} C_VEL
LIN {X 0,Y 559.163,Z 188.145,A -85,B 0,C 180,E1 -2858.624,E2 -2858.624} C_VEL
LIN {X 0,Y 559.152,Z 188.149,A -85,B 0,C 180,E1 -2860.926,E2 -2860.926} C_VEL
LIN {X 0,Y 559.154,Z 188.142,A -85,B 0,C 180,E1 -2863.948,E2 -2863.948} C_VEL
LIN {X 0,Y 559.159,Z 188.144,A -85,B 0,C 180,E1 -2866.184,E2 -2866.184} C_VEL
LIN {X 0,Y 559.198,Z 188.143,A -85,B 0,C 180,E1 -2868.605,E2 -2868.605} C_VEL
LIN {X 0,Y 559.161,Z 188.141,A -85,B 0,C 180,E1 -2871.325,E2 -2871.325} C_VEL
LIN {X 0,Y 559.218,Z 188.139,A -85,B 0,C 180,E1 -2874.23,E2 -2874.23} C_VEL
LIN {X 0,Y 559.239,Z 188.133,A -85,B 0,C 180,E1 -2877.839,E2 -2877.839} C_VEL
LIN {X 0,Y 559.27,Z 188.131,A -85,B 0,C 180,E1 -2880.72,E2 -2880.72} C_VEL
LIN {X 0,Y 559.234,Z 188.132,A -85,B 0,C 180,E1 -2882.881,E2 -2882.881} C_VEL
LIN {X 0,Y 559.219,Z 188.137,A -85,B 0,C 180,E1 -2885.77,E2 -2885.77} C_VEL
LIN {X 0,Y 559.185,Z 188.14,A -85,B 0,C 180,E1 -2888.674,E2 -2888.674} C_VEL
LIN {X 0,Y 559.198,Z 188.139,A -85,B 0,C 180,E1 -2891.601,E2 -2891.601} C_VEL
LIN {X 0,Y 559.193,Z 188.138,A -85,B 0,C 180,E1 -2894.596,E2 -2894.596} C_VEL
LIN {X 0,Y 559.157,Z 188.146,A -85,B 0,C 180,E1 -2897.557,E2 -2897.557} C_VEL
LIN {X 0,Y 559.166,Z 188.15,A -85,B 0,C 180,E1 -2899.838,E2 -2899.838} C_VEL
LIN {X 0,Y 559.135,Z 188.148,A -85,B 0,C 180,E1 -2902.153,E2 -2902.153} C_VEL
LIN {X 0,Y 559.173,Z 188.142,A -85,B 0,C 180,E1 -2905.188,E2 -2905.188} C_VEL
LIN {X 0,Y 559.189,Z 188.146,A -85,B 0,C 180,E1 -2907.712,E2 -2907.712} C_VEL
LIN {X 0,Y 559.157,Z 188.145,A -85,B 0,C 180,E1 -2911.019,E2 -2911.019} C_VEL
LIN {X 0,Y 559.171,Z 188.143,A -85,B 0,C 180,E1 -2913.951,E2 -2913.951} C_VEL
LIN {X 0,Y 559.135,Z 188.151,A -85,B 0,C 180,E1 -2917.109,E2 -2917.109} C_VEL
LIN {X 0,Y 559.163,Z 188.143,A -85,B 0,C 180,E1 -2919.943,E2 -2919.943} C_VEL
LIN {X 0,Y 559.152,Z 188.146,A -85,B 0,C 180,E1 -2922.744,E2 -2922.744} C_VEL
LIN {X 0,Y 559.145,Z 188.146,A -85,B 0,C 180,E1 -2925.761,E2 -2925.761} C_VEL
LIN {X 0,Y 559.158,Z 188.143,A -85,B 0,C 180,E1 -2928.23,E2 -2928.23} C_VEL
LIN {X 0,Y 559.171,Z 188.147,A -85,B 0,C 180,E1 -2931.192,E2 -2931.192} C_VEL
LIN {X 0,Y 559.134,Z 188.146,A -85,B 0,C 180,E1 -2933.79,E2 -2933.79} C_VEL
LIN {X 0,Y 559.158,Z 188.145,A -85,B 0,C 180,E1 -2936.426,E2 -2936.426} C_VEL
LIN {X 0,Y 559.151,Z 188.151,A -85,B 0,C 180,E1 -2938.981,E2 -2938.981} C_VEL
LIN {X 0,Y 559.177,Z 188.166,A -85,B 0,C 180,E1 -2941.421,E2 -2941.421} C_VEL
LIN {X 0,Y 562.2,Z 199.07,A -85,B 0,C 180,E1 -2942.568,E2 -2942.568} C_VEL
LIN {X 0,Y 561.729,Z 226.76,A -85,B 0,C 180,E1 -2945.023,E2 -2945.023} C_VEL
LIN {X 0,Y 561.583,Z 234.864,A -85,B 0,C 180,E1 -2945.733,E2 -2945.733} C_VEL
LIN {X 0,Y 563.204,Z 244.596,A -85,B 0,C 180,E1 -2945.942,E2 -2945.942} C_VEL
LIN {X 0,Y 562.299,Z 440.967,A -85,B 0,C 180,E1 -2948.581,E2 -2948.581} C_VEL
LIN {X 0,Y 562.098,Z 457.194,A -85,B 0,C 180,E1 -2948.933,E2 -2948.933} C_VEL
LIN {X 0,Y 561.764,Z 473.951,A -85,B 0,C 180,E1 -2949.447,E2 -2949.447} C_VEL
LIN {X 0,Y 561.494,Z 490.024,A -85,B 0,C 180,E1 -2950.101,E2 -2950.101} C_VEL
LIN {X 0,Y 561.137,Z 504.045,A -85,B 0,C 180,E1 -2950.806,E2 -2950.806} C_VEL
LIN {X 0,Y 560.764,Z 519.279,A -85,B 0,C 180,E1 -2951.741,E2 -2951.741} C_VEL
LIN {X 0,Y 560.366,Z 533.22,A -85,B 0,C 180,E1 -2952.765,E2 -2952.765} C_VEL
LIN {X 0,Y 559.997,Z 547.071,A -85,B 0,C 180,E1 -2953.973,E2 -2953.973} C_VEL
LIN {X 0,Y 559.659,Z 559.253,A -85,B 0,C 180,E1 -2955.225,E2 -2955.225} C_VEL
LIN {X 0,Y 559.429,Z 570.341,A -85,B 0,C 180,E1 -2956.561,E2 -2956.561} C_VEL
LIN {X 0,Y 559.219,Z 580.674,A -85,B 0,C 180,E1 -2958.032,E2 -2958.032} C_VEL
LIN {X 0,Y 559.073,Z 589.285,A -85,B 0,C 180,E1 -2959.498,E2 -2959.498} C_VEL
LIN {X 0,Y 558.937,Z 596.491,A -85,B 0,C 180,E1 -2960.957,E2 -2960.957} C_VEL
LIN {X 0,Y 558.893,Z 602.467,A -85,B 0,C 180,E1 -2962.413,E2 -2962.413} C_VEL
LIN {X 0,Y 558.864,Z 608.249,A -85,B 0,C 180,E1 -2964.226,E2 -2964.226} C_VEL
LIN {X 0,Y 558.805,Z 611.636,A -85,B 0,C 180,E1 -2965.673,E2 -2965.673} C_VEL
LIN {X 0,Y 558.787,Z 614.09,A -85,B 0,C 180,E1 -2967.117,E2 -2967.117} C_VEL
LIN {X 0,Y 558.739,Z 615.48,A -85,B 0,C 180,E1 -2968.559,E2 -2968.559} C_VEL
LIN {X 0,Y 558.735,Z 616,A -85,B 0,C 180,E1 -2970,E2 -2970} C_VEL
LIN {X 0,Y 558.739,Z 615.479,A -85,B 0,C 180,E1 -2971.442,E2 -2971.442} C_VEL
LIN {X 0,Y 558.787,Z 614.088,A -85,B 0,C 180,E1 -2972.884,E2 -2972.884} C_VEL
LIN {X 0,Y 558.805,Z 611.635,A -85,B 0,C 180,E1 -2974.328,E2 -2974.328} C_VEL
LIN {X 0,Y 558.863,Z 608.25,A -85,B 0,C 180,E1 -2975.774,E2 -2975.774} C_VEL
LIN {X 0,Y 558.893,Z 602.467,A -85,B 0,C 180,E1 -2977.587,E2 -2977.587} C_VEL
LIN {X 0,Y 558.93,Z 594.856,A -85,B 0,C 180,E1 -2979.408,E2 -2979.408} C_VEL
LIN {X 0,Y 559.116,Z 586.281,A -85,B 0,C 180,E1 -2981.046,E2 -2981.046} C_VEL
LIN {X 0,Y 559.275,Z 576.976,A -85,B 0,C 180,E1 -2982.519,E2 -2982.519} C_VEL
LIN {X 0,Y 559.472,Z 567.421,A -85,B 0,C 180,E1 -2983.808,E2 -2983.808} C_VEL
LIN {X 0,Y 559.791,Z 556.259,A -85,B 0,C 180,E1 -2985.103,E2 -2985.103} C_VEL
LIN {X 0,Y 560.05,Z 544.14,A -85,B 0,C 180,E1 -2986.307,E2 -2986.307} C_VEL
LIN {X 0,Y 560.42,Z 530.868,A -85,B 0,C 180,E1 -2987.422,E2 -2987.422} C_VEL
LIN {X 0,Y 560.808,Z 516.418,A -85,B 0,C 180,E1 -2988.447,E2 -2988.447} C_VEL
LIN {X 0,Y 561.19,Z 502.274,A -85,B 0,C 180,E1 -2989.287,E2 -2989.287} C_VEL
LIN {X 0,Y 561.546,Z 487.537,A -85,B 0,C 180,E1 -2990.014,E2 -2990.014} C_VEL
LIN {X 0,Y 561.85,Z 471.342,A -85,B 0,C 180,E1 -2990.646,E2 -2990.646} C_VEL
LIN {X 0,Y 562.138,Z 455.351,A -85,B 0,C 180,E1 -2991.114,E2 -2991.114} C_VEL
LIN {X 0,Y 562.261,Z 439.436,A -85,B 0,C 180,E1 -2991.445,E2 -2991.445} C_VEL
LIN {X 0,Y 563.192,Z 244.014,A -85,B 0,C 180,E1 -2994.067,E2 -2994.067} C_VEL
LIN {X 0,Y 561.602,Z 234.889,A -85,B 0,C 180,E1 -2994.266,E2 -2994.266} C_VEL
LIN {X 0,Y 562.257,Z 201.318,A -85,B 0,C 180,E1 -2997.231,E2 -2997.231} C_VEL
LIN {X 0,Y 561.971,Z 197.814,A -85,B 0,C 180,E1 -2997.563,E2 -2997.563} C_VEL
LIN {X 0,Y 559.17,Z 188.148,A -85,B 0,C 180,E1 -2998.606,E2 -2998.606} C_VEL
LIN {X 0,Y 559.159,Z 188.142,A -85,B 0,C 180,E1 -3001.863,E2 -3001.863} C_VEL
LIN {X 0,Y 559.137,Z 188.146,A -85,B 0,C 180,E1 -3004.445,E2 -3004.445} C_VEL
LIN {X 0,Y 559.131,Z 188.148,A -85,B 0,C 180,E1 -3007.639,E2 -3007.639} C_VEL
LIN {X 0,Y 559.159,Z 188.14,A -85,B 0,C 180,E1 -3009.942,E2 -3009.942} C_VEL
LIN {X 0,Y 559.145,Z 188.148,A -85,B 0,C 180,E1 -3012.745,E2 -3012.745} C_VEL
LIN {X 0,Y 559.125,Z 188.15,A -85,B 0,C 180,E1 -3015.26,E2 -3015.26} C_VEL
LIN {X 0,Y 559.158,Z 188.142,A -85,B 0,C 180,E1 -3018.229,E2 -3018.229} C_VEL
LIN {X 0,Y 559.169,Z 188.146,A -85,B 0,C 180,E1 -3021.192,E2 -3021.192} C_VEL
LIN {X 0,Y 559.135,Z 188.142,A -85,B 0,C 180,E1 -3023.789,E2 -3023.789} C_VEL
LIN {X 0,Y 559.144,Z 188.147,A -85,B 0,C 180,E1 -3026.424,E2 -3026.424} C_VEL
LIN {X 0,Y 559.153,Z 188.148,A -85,B 0,C 180,E1 -3028.981,E2 -3028.981} C_VEL
LIN {X 0,Y 559.141,Z 188.143,A -85,B 0,C 180,E1 -3031.623,E2 -3031.623} C_VEL
LIN {X 0,Y 559.173,Z 188.136,A -85,B 0,C 180,E1 -3033.903,E2 -3033.903} C_VEL
LIN {X 0,Y 559.137,Z 188.151,A -85,B 0,C 180,E1 -3036.571,E2 -3036.571} C_VEL
LIN {X 0,Y 559.171,Z 188.137,A -85,B 0,C 180,E1 -3039.395,E2 -3039.395} C_VEL
LIN {X 0,Y 559.135,Z 188.14,A -85,B 0,C 180,E1 -3041.685,E2 -3041.685} C_VEL
LIN {X 0,Y 559.159,Z 188.142,A -85,B 0,C 180,E1 -3043.948,E2 -3043.948} C_VEL
LIN {X 0,Y 559.163,Z 188.145,A -85,B 0,C 180,E1 -3046.184,E2 -3046.184} C_VEL
LIN {X 0,Y 559.202,Z 188.138,A -85,B 0,C 180,E1 -3048.605,E2 -3048.605} C_VEL
LIN {X 0,Y 559.165,Z 188.14,A -85,B 0,C 180,E1 -3051.325,E2 -3051.325} C_VEL
LIN {X 0,Y 559.221,Z 188.14,A -85,B 0,C 180,E1 -3054.23,E2 -3054.23} C_VEL
LIN {X 0,Y 559.241,Z 188.126,A -85,B 0,C 180,E1 -3057.839,E2 -3057.839} C_VEL
LIN {X 0,Y 559.272,Z 188.13,A -85,B 0,C 180,E1 -3060.72,E2 -3060.72} C_VEL
LIN {X 0,Y 559.236,Z 188.132,A -85,B 0,C 180,E1 -3062.881,E2 -3062.881} C_VEL
LIN {X 0,Y 559.221,Z 188.132,A -85,B 0,C 180,E1 -3065.77,E2 -3065.77} C_VEL
LIN {X 0,Y 559.182,Z 188.14,A -85,B 0,C 180,E1 -3068.674,E2 -3068.674} C_VEL
LIN {X 0,Y 559.202,Z 188.135,A -85,B 0,C 180,E1 -3071.6,E2 -3071.6} C_VEL
LIN {X 0,Y 559.197,Z 188.138,A -85,B 0,C 180,E1 -3074.596,E2 -3074.596} C_VEL
LIN {X 0,Y 559.16,Z 188.143,A -85,B 0,C 180,E1 -3077.557,E2 -3077.557} C_VEL
LIN {X 0,Y 559.169,Z 188.144,A -85,B 0,C 180,E1 -3079.837,E2 -3079.837} C_VEL
LIN {X 0,Y 559.138,Z 188.149,A -85,B 0,C 180,E1 -3082.153,E2 -3082.153} C_VEL
LIN {X 0,Y 559.176,Z 188.137,A -85,B 0,C 180,E1 -3085.187,E2 -3085.187} C_VEL
LIN {X 0,Y 559.189,Z 188.144,A -85,B 0,C 180,E1 -3087.712,E2 -3087.712} C_VEL
LIN {X 0,Y 559.144,Z 188.142,A -85,B 0,C 180,E1 -3090.622,E2 -3090.622} C_VEL
LIN {X 0,Y 558.479,Z 188.228,A -85,B 0,C 180,E1 -3091.223,E2 -3091.223} C_VEL
LIN {X 0,Y 555.616,Z 188.583,A -85,B 0,C 180,E1 -3092.199,E2 -3092.199} C_VEL
LIN {X 0,Y 553.206,Z 188.881,A -85,B 0,C 180,E1 -3092.985,E2 -3092.985} C_VEL
LIN {X 0,Y 552.187,Z 189.015,A -85,B 0,C 180,E1 -3093.592,E2 -3093.592} C_VEL
LIN {X 0,Y 552.113,Z 189.02,A -85,B 0,C 180,E1 -3093.797,E2 -3093.797} C_VEL
LIN {X 0,Y 552.109,Z 189.018,A -85,B 0,C 180,E1 -3096.747,E2 -3096.747} C_VEL
LIN {X 0,Y 552.127,Z 189.023,A -85,B 0,C 180,E1 -3099.527,E2 -3099.527} C_VEL
LIN {X 0,Y 552.128,Z 189.016,A -85,B 0,C 180,E1 -3102.425,E2 -3102.425} C_VEL
LIN {X 0,Y 552.095,Z 189.03,A -85,B 0,C 180,E1 -3105.563,E2 -3105.563} C_VEL
LIN {X 0,Y 552.12,Z 189.016,A -85,B 0,C 180,E1 -3108.554,E2 -3108.554} C_VEL
LIN {X 0,Y 552.115,Z 189.028,A -85,B 0,C 180,E1 -3111.411,E2 -3111.411} C_VEL
LIN {X 0,Y 552.085,Z 189.02,A -85,B 0,C 180,E1 -3114.157,E2 -3114.157} C_VEL
LIN {X 0,Y 552.122,Z 189.021,A -85,B 0,C 180,E1 -3116.815,E2 -3116.815} C_VEL
LIN {X 0,Y 552.104,Z 189.028,A -85,B 0,C 180,E1 -3119.391,E2 -3119.391} C_VEL
LIN {X 0,Y 552.108,Z 189.019,A -85,B 0,C 180,E1 -3121.902,E2 -3121.902} C_VEL
LIN {X 0,Y 552.155,Z 189.016,A -85,B 0,C 180,E1 -3124.65,E2 -3124.65} C_VEL
LIN {X 0,Y 552.092,Z 189.026,A -85,B 0,C 180,E1 -3127.549,E2 -3127.549} C_VEL
LIN {X 0,Y 552.144,Z 189.012,A -85,B 0,C 180,E1 -3130.375,E2 -3130.375} C_VEL
LIN {X 0,Y 552.154,Z 189.021,A -85,B 0,C 180,E1 -3132.977,E2 -3132.977} C_VEL
LIN {X 0,Y 552.136,Z 189.011,A -85,B 0,C 180,E1 -3136.004,E2 -3136.004} C_VEL
LIN {X 0,Y 552.162,Z 189.021,A -85,B 0,C 180,E1 -3138.993,E2 -3138.993} C_VEL
LIN {X 0,Y 552.158,Z 189.015,A -85,B 0,C 180,E1 -3141.951,E2 -3141.951} C_VEL
LIN {X 0,Y 552.226,Z 189.014,A -85,B 0,C 180,E1 -3144.889,E2 -3144.889} C_VEL
LIN {X 0,Y 552.225,Z 189.008,A -85,B 0,C 180,E1 -3147.812,E2 -3147.812} C_VEL
LIN {X 0,Y 552.229,Z 189.049,A -85,B 0,C 180,E1 -3149.544,E2 -3149.544} C_VEL
LIN {X 0,Y 554.774,Z 199.041,A -85,B 0,C 180,E1 -3150.726,E2 -3150.726} C_VEL
LIN {X 0,Y 554.723,Z 206.257,A -85,B 0,C 180,E1 -3151.47,E2 -3151.47} C_VEL
LIN {X 0,Y 556.73,Z 216.157,A -85,B 0,C 180,E1 -3151.705,E2 -3151.705} C_VEL
LIN {X 0,Y 555.682,Z 410.517,A -85,B 0,C 180,E1 -3154.352,E2 -3154.352} C_VEL
LIN {X 0,Y 555.483,Z 426.516,A -85,B 0,C 180,E1 -3154.694,E2 -3154.694} C_VEL
LIN {X 0,Y 555.147,Z 442.444,A -85,B 0,C 180,E1 -3155.175,E2 -3155.175} C_VEL
LIN {X 0,Y 554.769,Z 458.373,A -85,B 0,C 180,E1 -3155.816,E2 -3155.816} C_VEL
LIN {X 0,Y 554.425,Z 472.927,A -85,B 0,C 180,E1 -3156.551,E2 -3156.551} C_VEL
LIN {X 0,Y 553.978,Z 487.307,A -85,B 0,C 180,E1 -3157.421,E2 -3157.421} C_VEL
LIN {X 0,Y 553.574,Z 501.611,A -85,B 0,C 180,E1 -3158.459,E2 -3158.459} C_VEL
LIN {X 0,Y 553.181,Z 513.868,A -85,B 0,C 180,E1 -3159.506,E2 -3159.506} C_VEL
LIN {X 0,Y 552.847,Z 525.066,A -85,B 0,C 180,E1 -3160.622,E2 -3160.622} C_VEL
LIN {X 0,Y 552.527,Z 536.398,A -85,B 0,C 180,E1 -3161.928,E2 -3161.928} C_VEL
LIN {X 0,Y 552.296,Z 546.17,A -85,B 0,C 180,E1 -3163.241,E2 -3163.241} C_VEL
LIN {X 0,Y 552.083,Z 555.659,A -85,B 0,C 180,E1 -3164.749,E2 -3164.749} C_VEL
LIN {X 0,Y 551.886,Z 563.651,A -85,B 0,C 180,E1 -3166.269,E2 -3166.269} C_VEL
LIN {X 0,Y 551.813,Z 570.311,A -85,B 0,C 180,E1 -3167.798,E2 -3167.798} C_VEL
LIN {X 0,Y 551.747,Z 576.266,A -85,B 0,C 180,E1 -3169.509,E2 -3169.509} C_VEL
LIN {X 0,Y 551.665,Z 579.982,A -85,B 0,C 180,E1 -3170.898,E2 -3170.898} C_VEL
LIN {X 0,Y 551.642,Z 583.097,A -85,B 0,C 180,E1 -3172.47,E2 -3172.47} C_VEL
LIN {X 0,Y 551.593,Z 585.114,A -85,B 0,C 180,E1 -3174.061,E2 -3174.061} C_VEL
LIN {X 0,Y 551.62,Z 585.926,A -85,B 0,C 180,E1 -3175.669,E2 -3175.669} C_VEL
LIN {X 0,Y 551.622,Z 585.611,A -85,B 0,C 180,E1 -3177.3,E2 -3177.3} C_VEL
LIN {X 0,Y 551.643,Z 584.105,A -85,B 0,C 180,E1 -3178.954,E2 -3178.954} C_VEL
LIN {X 0,Y 551.69,Z 581.23,A -85,B 0,C 180,E1 -3180.634,E2 -3180.634} C_VEL
LIN {X 0,Y 551.722,Z 576.948,A -85,B 0,C 180,E1 -3182.344,E2 -3182.344} C_VEL
LIN {X 0,Y 551.808,Z 570.965,A -85,B 0,C 180,E1 -3184.121,E2 -3184.121} C_VEL
LIN {X 0,Y 551.891,Z 564.689,A -85,B 0,C 180,E1 -3185.606,E2 -3185.606} C_VEL
LIN {X 0,Y 552.027,Z 556.436,A -85,B 0,C 180,E1 -3187.209,E2 -3187.209} C_VEL
LIN {X 0,Y 552.26,Z 546.305,A -85,B 0,C 180,E1 -3188.83,E2 -3188.83} C_VEL
LIN {X 0,Y 552.525,Z 535.674,A -85,B 0,C 180,E1 -3190.254,E2 -3190.254} C_VEL
LIN {X 0,Y 552.845,Z 524.886,A -85,B 0,C 180,E1 -3191.488,E2 -3191.488} C_VEL
LIN {X 0,Y 553.269,Z 511.919,A -85,B 0,C 180,E1 -3192.757,E2 -3192.757} C_VEL
LIN {X 0,Y 553.642,Z 499.327,A -85,B 0,C 180,E1 -3193.811,E2 -3193.811} C_VEL
LIN {X 0,Y 554.057,Z 484.809,A -85,B 0,C 180,E1 -3194.837,E2 -3194.837} C_VEL
LIN {X 0,Y 554.48,Z 469.864,A -85,B 0,C 180,E1 -3195.709,E2 -3195.709} C_VEL
LIN {X 0,Y 554.9,Z 454.357,A -85,B 0,C 180,E1 -3196.446,E2 -3196.446} C_VEL
LIN {X 0,Y 555.237,Z 437.937,A -85,B 0,C 180,E1 -3197.063,E2 -3197.063} C_VEL
LIN {X 0,Y 555.543,Z 421.408,A -85,B 0,C 180,E1 -3197.521,E2 -3197.521} C_VEL
LIN {X 0,Y 555.764,Z 404.453,A -85,B 0,C 180,E1 -3197.835,E2 -3197.835} C_VEL
LIN {X 0,Y 556.679,Z 216.843,A -85,B 0,C 180,E1 -3200.379,E2 -3200.379} C_VEL
LIN {X 0,Y 554.722,Z 206.32,A -85,B 0,C 180,E1 -3200.624,E2 -3200.624} C_VEL
LIN {X 0,Y 554.694,Z 198.937,A -85,B 0,C 180,E1 -3201.391,E2 -3201.391} C_VEL
LIN {X 0,Y 552.074,Z 189.031,A -85,B 0,C 180,E1 -3202.594,E2 -3202.594} C_VEL
LIN {X 0,Y 552.116,Z 189.021,A -85,B 0,C 180,E1 -3205.831,E2 -3205.831} C_VEL
LIN {X 0,Y 552.113,Z 189.023,A -85,B 0,C 180,E1 -3208.54,E2 -3208.54} C_VEL
LIN {X 0,Y 552.087,Z 189.027,A -85,B 0,C 180,E1 -3211.443,E2 -3211.443} C_VEL
LIN {X 0,Y 552.073,Z 189.026,A -85,B 0,C 180,E1 -3214.353,E2 -3214.353} C_VEL
LIN {X 0,Y 552.084,Z 189.03,A -85,B 0,C 180,E1 -3216.757,E2 -3216.757} C_VEL
LIN {X 0,Y 552.109,Z 189.026,A -85,B 0,C 180,E1 -3219.119,E2 -3219.119} C_VEL
LIN {X 0,Y 552.11,Z 189.021,A -85,B 0,C 180,E1 -3221.444,E2 -3221.444} C_VEL
LIN {X 0,Y 552.105,Z 189.02,A -85,B 0,C 180,E1 -3223.737,E2 -3223.737} C_VEL
LIN {X 0,Y 552.124,Z 189.019,A -85,B 0,C 180,E1 -3226.004,E2 -3226.004} C_VEL
LIN {X 0,Y 552.153,Z 189.018,A -85,B 0,C 180,E1 -3228.993,E2 -3228.993} C_VEL
LIN {X 0,Y 552.143,Z 189.017,A -85,B 0,C 180,E1 -3231.951,E2 -3231.951} C_VEL
LIN {X 0,Y 552.217,Z 189.009,A -85,B 0,C 180,E1 -3234.889,E2 -3234.889} C_VEL
LIN {X 0,Y 552.212,Z 189.009,A -85,B 0,C 180,E1 -3237.812,E2 -3237.812} C_VEL
LIN {X 0,Y 552.239,Z 189.006,A -85,B 0,C 180,E1 -3240.729,E2 -3240.729} C_VEL
LIN {X 0,Y 552.2,Z 189.008,A -85,B 0,C 180,E1 -3242.918,E2 -3242.918} C_VEL
LIN {X 0,Y 552.189,Z 189.014,A -85,B 0,C 180,E1 -3245.844,E2 -3245.844} C_VEL
LIN {X 0,Y 552.156,Z 189.014,A -85,B 0,C 180,E1 -3248.786,E2 -3248.786} C_VEL
LIN {X 0,Y 552.156,Z 189.018,A -85,B 0,C 180,E1 -3251.751,E2 -3251.751} C_VEL
LIN {X 0,Y 552.13,Z 189.017,A -85,B 0,C 180,E1 -3254.749,E2 -3254.749} C_VEL
LIN {X 0,Y 552.108,Z 189.028,A -85,B 0,C 180,E1 -3257.788,E2 -3257.788} C_VEL
LIN {X 0,Y 552.124,Z 189.023,A -85,B 0,C 180,E1 -3260.101,E2 -3260.101} C_VEL
LIN {X 0,Y 552.089,Z 189.023,A -85,B 0,C 180,E1 -3262.451,E2 -3262.451} C_VEL
LIN {X 0,Y 552.151,Z 189.019,A -85,B 0,C 180,E1 -3265.351,E2 -3265.351} C_VEL
LIN {X 0,Y 552.12,Z 189.021,A -85,B 0,C 180,E1 -3268.098,E2 -3268.098} C_VEL
LIN {X 0,Y 552.101,Z 189.021,A -85,B 0,C 180,E1 -3270.609,E2 -3270.609} C_VEL
LIN {X 0,Y 552.123,Z 189.024,A -85,B 0,C 180,E1 -3273.185,E2 -3273.185} C_VEL
LIN {X 0,Y 552.083,Z 189.027,A -85,B 0,C 180,E1 -3275.844,E2 -3275.844} C_VEL
LIN {X 0,Y 552.119,Z 189.025,A -85,B 0,C 180,E1 -3279.062,E2 -3279.062} C_VEL
LIN {X 0,Y 552.123,Z 189.026,A -85,B 0,C 180,E1 -3281.446,E2 -3281.446} C_VEL
LIN {X 0,Y 552.089,Z 189.025,A -85,B 0,C 180,E1 -3284.532,E2 -3284.532} C_VEL
LIN {X 0,Y 552.124,Z 189.022,A -85,B 0,C 180,E1 -3287.585,E2 -3287.585} C_VEL
LIN {X 0,Y 552.128,Z 189.021,A -85,B 0,C 180,E1 -3290.474,E2 -3290.474} C_VEL
LIN {X 0,Y 552.102,Z 189.026,A -85,B 0,C 180,E1 -3293.317,E2 -3293.317} C_VEL
LIN {X 0,Y 552.122,Z 189.018,A -85,B 0,C 180,E1 -3295.939,E2 -3295.939} C_VEL
LIN {X 0,Y 552.115,Z 189.024,A -85,B 0,C 180,E1 -3298.541,E2 -3298.541} C_VEL
LIN {X 0,Y 552.107,Z 189.069,A -85,B 0,C 180,E1 -3301.126,E2 -3301.126} C_VEL
LIN {X 0,Y 555.587,Z 201.311,A -85,B 0,C 180,E1 -3302.439,E2 -3302.439} C_VEL
LIN {X 0,Y 554.919,Z 232.105,A -85,B 0,C 180,E1 -3305.196,E2 -3305.196} C_VEL
LIN {X 0,Y 554.85,Z 234.629,A -85,B 0,C 180,E1 -3305.419,E2 -3305.419} C_VEL
LIN {X 0,Y 556.7,Z 245.014,A -85,B 0,C 180,E1 -3305.652,E2 -3305.652} C_VEL
LIN {X 0,Y 555.685,Z 440.852,A -85,B 0,C 180,E1 -3308.313,E2 -3308.313} C_VEL
LIN {X 0,Y 555.464,Z 457.152,A -85,B 0,C 180,E1 -3308.669,E2 -3308.669} C_VEL
LIN {X 0,Y 555.117,Z 473.95,A -85,B 0,C 180,E1 -3309.19,E2 -3309.19} C_VEL
LIN {X 0,Y 554.82,Z 488.414,A -85,B 0,C 180,E1 -3309.774,E2 -3309.774} C_VEL
LIN {X 0,Y 554.39,Z 504.049,A -85,B 0,C 180,E1 -3310.563,E2 -3310.563} C_VEL
LIN {X 0,Y 553.96,Z 519.276,A -85,B 0,C 180,E1 -3311.509,E2 -3311.509} C_VEL
LIN {X 0,Y 553.473,Z 533.36,A -85,B 0,C 180,E1 -3312.555,E2 -3312.555} C_VEL
LIN {X 0,Y 553.046,Z 547.07,A -85,B 0,C 180,E1 -3313.766,E2 -3313.766} C_VEL
LIN {X 0,Y 552.757,Z 558.3,A -85,B 0,C 180,E1 -3314.926,E2 -3314.926} C_VEL
LIN {X 0,Y 552.445,Z 568.908,A -85,B 0,C 180,E1 -3316.201,E2 -3316.201} C_VEL
LIN {X 0,Y 552.208,Z 579.442,A -85,B 0,C 180,E1 -3317.692,E2 -3317.692} C_VEL
LIN {X 0,Y 551.992,Z 588.277,A -85,B 0,C 180,E1 -3319.176,E2 -3319.176} C_VEL
LIN {X 0,Y 551.861,Z 594.857,A -85,B 0,C 180,E1 -3320.471,E2 -3320.471} C_VEL
LIN {X 0,Y 551.803,Z 602.467,A -85,B 0,C 180,E1 -3322.315,E2 -3322.315} C_VEL
LIN {X 0,Y 551.771,Z 608.25,A -85,B 0,C 180,E1 -3324.152,E2 -3324.152} C_VEL
LIN {X 0,Y 551.701,Z 611.636,A -85,B 0,C 180,E1 -3325.617,E2 -3325.617} C_VEL
LIN {X 0,Y 551.711,Z 614.09,A -85,B 0,C 180,E1 -3327.08,E2 -3327.08} C_VEL
LIN {X 0,Y 551.638,Z 615.479,A -85,B 0,C 180,E1 -3328.54,E2 -3328.54} C_VEL
LIN {X 0,Y 551.636,Z 616,A -85,B 0,C 180,E1 -3330,E2 -3330} C_VEL
LIN {X 0,Y 551.638,Z 615.479,A -85,B 0,C 180,E1 -3331.46,E2 -3331.46} C_VEL
LIN {X 0,Y 551.711,Z 614.089,A -85,B 0,C 180,E1 -3332.921,E2 -3332.921} C_VEL
LIN {X 0,Y 551.701,Z 611.634,A -85,B 0,C 180,E1 -3334.384,E2 -3334.384} C_VEL
LIN {X 0,Y 551.771,Z 608.25,A -85,B 0,C 180,E1 -3335.849,E2 -3335.849} C_VEL
LIN {X 0,Y 551.804,Z 602.467,A -85,B 0,C 180,E1 -3337.685,E2 -3337.685} C_VEL
LIN {X 0,Y 551.861,Z 594.856,A -85,B 0,C 180,E1 -3339.53,E2 -3339.53} C_VEL
LIN {X 0,Y 552.04,Z 587.267,A -85,B 0,C 180,E1 -3341.009,E2 -3341.009} C_VEL
LIN {X 0,Y 552.226,Z 578.209,A -85,B 0,C 180,E1 -3342.495,E2 -3342.495} C_VEL
LIN {X 0,Y 552.484,Z 567.421,A -85,B 0,C 180,E1 -3343.987,E2 -3343.987} C_VEL
LIN {X 0,Y 552.855,Z 556.448,A -85,B 0,C 180,E1 -3345.277,E2 -3345.277} C_VEL
LIN {X 0,Y 553.161,Z 544.138,A -85,B 0,C 180,E1 -3346.516,E2 -3346.516} C_VEL
LIN {X 0,Y 553.578,Z 530.635,A -85,B 0,C 180,E1 -3347.663,E2 -3347.663} C_VEL
LIN {X 0,Y 553.987,Z 516.415,A -85,B 0,C 180,E1 -3348.683,E2 -3348.683} C_VEL
LIN {X 0,Y 554.414,Z 502.27,A -85,B 0,C 180,E1 -3349.532,E2 -3349.532} C_VEL
LIN {X 0,Y 554.846,Z 487.262,A -85,B 0,C 180,E1 -3350.278,E2 -3350.278} C_VEL
LIN {X 0,Y 555.191,Z 471.341,A -85,B 0,C 180,E1 -3350.905,E2 -3350.905} C_VEL
LIN {X 0,Y 555.501,Z 455.308,A -85,B 0,C 180,E1 -3351.378,E2 -3351.378} C_VEL
LIN {X 0,Y 555.649,Z 439.327,A -85,B 0,C 180,E1 -3351.713,E2 -3351.713} C_VEL
LIN {X 0,Y 556.661,Z 244.301,A -85,B 0,C 180,E1 -3354.36,E2 -3354.36} C_VEL
LIN {X 0,Y 554.872,Z 234.631,A -85,B 0,C 180,E1 -3354.586,E2 -3354.586} C_VEL
LIN {X 0,Y 555.633,Z 201.518,A -85,B 0,C 180,E1 -3357.549,E2 -3357.549} C_VEL
LIN {X 0,Y 552.104,Z 189.029,A -85,B 0,C 180,E1 -3358.902,E2 -3358.902} C_VEL
LIN {X 0,Y 552.109,Z 189.025,A -85,B 0,C 180,E1 -3361.475,E2 -3361.475} C_VEL
LIN {X 0,Y 552.128,Z 189.019,A -85,B 0,C 180,E1 -3364.17,E2 -3364.17} C_VEL
LIN {X 0,Y 552.096,Z 189.026,A -85,B 0,C 180,E1 -3366.748,E2 -3366.748} C_VEL
LIN {X 0,Y 552.128,Z 189.02,A -85,B 0,C 180,E1 -3369.527,E2 -3369.527} C_VEL
LIN {X 0,Y 552.105,Z 189.022,A -85,B 0,C 180,E1 -3372.427,E2 -3372.427} C_VEL
LIN {X 0,Y 552.074,Z 189.024,A -85,B 0,C 180,E1 -3375.56,E2 -3375.56} C_VEL
LIN {X 0,Y 552.117,Z 189.024,A -85,B 0,C 180,E1 -3378.678,E2 -3378.678} C_VEL
LIN {X 0,Y 552.112,Z 189.022,A -85,B 0,C 180,E1 -3381.411,E2 -3381.411} C_VEL
LIN {X 0,Y 552.082,Z 189.021,A -85,B 0,C 180,E1 -3384.156,E2 -3384.156} C_VEL
LIN {X 0,Y 552.104,Z 189.028,A -85,B 0,C 180,E1 -3386.814,E2 -3386.814} C_VEL
LIN {X 0,Y 552.098,Z 189.021,A -85,B 0,C 180,E1 -3389.391,E2 -3389.391} C_VEL
LIN {X 0,Y 552.093,Z 189.022,A -85,B 0,C 180,E1 -3391.901,E2 -3391.901} C_VEL
LIN {X 0,Y 552.134,Z 189.02,A -85,B 0,C 180,E1 -3394.654,E2 -3394.654} C_VEL
LIN {X 0,Y 552.088,Z 189.022,A -85,B 0,C 180,E1 -3397.549,E2 -3397.549} C_VEL
LIN {X 0,Y 552.14,Z 189.018,A -85,B 0,C 180,E1 -3400.375,E2 -3400.375} C_VEL
LIN {X 0,Y 552.13,Z 189.02,A -85,B 0,C 180,E1 -3402.977,E2 -3402.977} C_VEL
LIN {X 0,Y 552.128,Z 189.019,A -85,B 0,C 180,E1 -3406.004,E2 -3406.004} C_VEL
LIN {X 0,Y 552.157,Z 189.011,A -85,B 0,C 180,E1 -3408.993,E2 -3408.993} C_VEL
LIN {X 0,Y 552.147,Z 189.017,A -85,B 0,C 180,E1 -3411.951,E2 -3411.951} C_VEL
LIN {X 0,Y 552.22,Z 189.004,A -85,B 0,C 180,E1 -3414.889,E2 -3414.889} C_VEL
LIN {X 0,Y 552.214,Z 189,A -85,B 0,C 180,E1 -3417.812,E2 -3417.812} C_VEL
LIN {X 0,Y 552.241,Z 189.006,A -85,B 0,C 180,E1 -3420.729,E2 -3420.729} C_VEL
LIN {X 0,Y 552.202,Z 189.008,A -85,B 0,C 180,E1 -3422.918,E2 -3422.918} C_VEL
LIN {X 0,Y 552.192,Z 189.008,A -85,B 0,C 180,E1 -3425.844,E2 -3425.844} C_VEL
LIN {X 0,Y 552.15,Z 189.015,A -85,B 0,C 180,E1 -3428.786,E2 -3428.786} C_VEL
LIN {X 0,Y 552.159,Z 189.014,A -85,B 0,C 180,E1 -3431.751,E2 -3431.751} C_VEL
LIN {X 0,Y 552.133,Z 189.017,A -85,B 0,C 180,E1 -3434.748,E2 -3434.748} C_VEL
LIN {X 0,Y 552.111,Z 189.024,A -85,B 0,C 180,E1 -3437.788,E2 -3437.788} C_VEL
LIN {X 0,Y 552.128,Z 189.023,A -85,B 0,C 180,E1 -3440.101,E2 -3440.101} C_VEL
LIN {X 0,Y 552.093,Z 189.023,A -85,B 0,C 180,E1 -3442.451,E2 -3442.451} C_VEL
LIN {X 0,Y 552.153,Z 189.013,A -85,B 0,C 180,E1 -3445.351,E2 -3445.351} C_VEL
LIN {X 0,Y 552.123,Z 189.023,A -85,B 0,C 180,E1 -3448.097,E2 -3448.097} C_VEL
LIN {X 0,Y 552.106,Z 189.018,A -85,B 0,C 180,E1 -3450.617,E2 -3450.617} C_VEL
LIN {X 0,Y 552.12,Z 189.017,A -85,B 0,C 180,E1 -3453.185,E2 -3453.185} C_VEL
LIN {X 0,Y 552.113,Z 189.02,A -85,B 0,C 180,E1 -3453.797,E2 -3453.797} C_VEL
LIN {X 0,Y 551.477,Z 189.103,A -85,B 0,C 180,E1 -3454.406,E2 -3454.406} C_VEL
LIN {X 0,Y 548.656,Z 189.454,A -85,B 0,C 180,E1 -3455.394,E2 -3455.394} C_VEL
LIN {X 0,Y 546.235,Z 189.752,A -85,B 0,C 180,E1 -3456.189,E2 -3456.189} C_VEL
LIN {X 0,Y 545.165,Z 189.884,A -85,B 0,C 180,E1 -3456.803,E2 -3456.803} C_VEL
LIN {X 0,Y 545.062,Z 189.897,A -85,B 0,C 180,E1 -3457.011,E2 -3457.011} C_VEL
LIN {X 0,Y 545.064,Z 189.899,A -85,B 0,C 180,E1 -3460.143,E2 -3460.143} C_VEL
LIN {X 0,Y 545.076,Z 189.897,A -85,B 0,C 180,E1 -3463.107,E2 -3463.107} C_VEL
LIN {X 0,Y 545.065,Z 189.898,A -85,B 0,C 180,E1 -3466.224,E2 -3466.224} C_VEL
LIN {X 0,Y 545.08,Z 189.895,A -85,B 0,C 180,E1 -3468.886,E2 -3468.886} C_VEL
LIN {X 0,Y 545.05,Z 189.902,A -85,B 0,C 180,E1 -3471.763,E2 -3471.763} C_VEL
LIN {X 0,Y 545.037,Z 189.898,A -85,B 0,C 180,E1 -3474.532,E2 -3474.532} C_VEL
LIN {X 0,Y 545.08,Z 189.903,A -85,B 0,C 180,E1 -3477.213,E2 -3477.213} C_VEL
LIN {X 0,Y 545.064,Z 189.9,A -85,B 0,C 180,E1 -3479.811,E2 -3479.811} C_VEL
LIN {X 0,Y 545.08,Z 189.894,A -85,B 0,C 180,E1 -3482.344,E2 -3482.344} C_VEL
LIN {X 0,Y 545.117,Z 189.895,A -85,B 0,C 180,E1 -3484.821,E2 -3484.821} C_VEL
LIN {X 0,Y 545.038,Z 189.909,A -85,B 0,C 180,E1 -3487.242,E2 -3487.242} C_VEL
LIN {X 0,Y 545.115,Z 189.888,A -85,B 0,C 180,E1 -3490.415,E2 -3490.415} C_VEL
LIN {X 0,Y 545.069,Z 189.901,A -85,B 0,C 180,E1 -3493.521,E2 -3493.521} C_VEL
LIN {X 0,Y 545.095,Z 189.888,A -85,B 0,C 180,E1 -3495.82,E2 -3495.82} C_VEL
LIN {X 0,Y 545.118,Z 189.899,A -85,B 0,C 180,E1 -3498.849,E2 -3498.849} C_VEL
LIN {X 0,Y 545.128,Z 189.891,A -85,B 0,C 180,E1 -3501.847,E2 -3501.847} C_VEL
LIN {X 0,Y 545.203,Z 189.888,A -85,B 0,C 180,E1 -3504.823,E2 -3504.823} C_VEL
LIN {X 0,Y 545.196,Z 189.884,A -85,B 0,C 180,E1 -3507.784,E2 -3507.784} C_VEL
LIN {X 0,Y 545.209,Z 190.028,A -85,B 0,C 180,E1 -3509.261,E2 -3509.261} C_VEL
LIN {X 0,Y 548.006,Z 200.739,A -85,B 0,C 180,E1 -3510.551,E2 -3510.551} C_VEL
LIN {X 0,Y 548.053,Z 206.337,A -85,B 0,C 180,E1 -3511.139,E2 -3511.139} C_VEL
LIN {X 0,Y 550.273,Z 217.232,A -85,B 0,C 180,E1 -3511.413,E2 -3511.413} C_VEL
LIN {X 0,Y 549.097,Z 412.098,A -85,B 0,C 180,E1 -3514.105,E2 -3514.105} C_VEL
LIN {X 0,Y 548.862,Z 428.428,A -85,B 0,C 180,E1 -3514.475,E2 -3514.475} C_VEL
LIN {X 0,Y 548.459,Z 443.945,A -85,B 0,C 180,E1 -3514.962,E2 -3514.962} C_VEL
LIN {X 0,Y 548.07,Z 459.661,A -85,B 0,C 180,E1 -3515.611,E2 -3515.611} C_VEL
LIN {X 0,Y 547.576,Z 475.699,A -85,B 0,C 180,E1 -3516.448,E2 -3516.448} C_VEL
LIN {X 0,Y 547.149,Z 490.232,A -85,B 0,C 180,E1 -3517.38,E2 -3517.38} C_VEL
LIN {X 0,Y 546.686,Z 503.623,A -85,B 0,C 180,E1 -3518.399,E2 -3518.399} C_VEL
LIN {X 0,Y 546.24,Z 515.459,A -85,B 0,C 180,E1 -3519.441,E2 -3519.441} C_VEL
LIN {X 0,Y 545.83,Z 528.194,A -85,B 0,C 180,E1 -3520.76,E2 -3520.76} C_VEL
LIN {X 0,Y 545.49,Z 539.035,A -85,B 0,C 180,E1 -3522.085,E2 -3522.085} C_VEL
LIN {X 0,Y 545.225,Z 548.4,A -85,B 0,C 180,E1 -3523.416,E2 -3523.416} C_VEL
LIN {X 0,Y 545.002,Z 557.568,A -85,B 0,C 180,E1 -3524.945,E2 -3524.945} C_VEL
LIN {X 0,Y 544.824,Z 565.29,A -85,B 0,C 180,E1 -3526.486,E2 -3526.486} C_VEL
LIN {X 0,Y 544.718,Z 571.624,A -85,B 0,C 180,E1 -3528.038,E2 -3528.038} C_VEL
LIN {X 0,Y 544.669,Z 576.828,A -85,B 0,C 180,E1 -3529.621,E2 -3529.621} C_VEL
LIN {X 0,Y 544.589,Z 580.812,A -85,B 0,C 180,E1 -3531.182,E2 -3531.182} C_VEL
LIN {X 0,Y 544.529,Z 583.633,A -85,B 0,C 180,E1 -3532.78,E2 -3532.78} C_VEL
LIN {X 0,Y 544.511,Z 585.368,A -85,B 0,C 180,E1 -3534.394,E2 -3534.394} C_VEL
LIN {X 0,Y 544.55,Z 585.999,A -85,B 0,C 180,E1 -3536.027,E2 -3536.027} C_VEL
LIN {X 0,Y 544.54,Z 585.375,A -85,B 0,C 180,E1 -3537.685,E2 -3537.685} C_VEL
LIN {X 0,Y 544.551,Z 583.547,A -85,B 0,C 180,E1 -3539.368,E2 -3539.368} C_VEL
LIN {X 0,Y 544.606,Z 580.418,A -85,B 0,C 180,E1 -3541.076,E2 -3541.076} C_VEL
LIN {X 0,Y 544.636,Z 577.083,A -85,B 0,C 180,E1 -3542.378,E2 -3542.378} C_VEL
LIN {X 0,Y 544.723,Z 571.747,A -85,B 0,C 180,E1 -3544.019,E2 -3544.019} C_VEL
LIN {X 0,Y 544.812,Z 565.121,A -85,B 0,C 180,E1 -3545.641,E2 -3545.641} C_VEL
LIN {X 0,Y 544.968,Z 556.692,A -85,B 0,C 180,E1 -3547.309,E2 -3547.309} C_VEL
LIN {X 0,Y 545.178,Z 548.255,A -85,B 0,C 180,E1 -3548.698,E2 -3548.698} C_VEL
LIN {X 0,Y 545.488,Z 538.271,A -85,B 0,C 180,E1 -3550.104,E2 -3550.104} C_VEL
LIN {X 0,Y 545.821,Z 526.552,A -85,B 0,C 180,E1 -3551.51,E2 -3551.51} C_VEL
LIN {X 0,Y 546.268,Z 515.267,A -85,B 0,C 180,E1 -3552.667,E2 -3552.667} C_VEL
LIN {X 0,Y 546.675,Z 502.37,A -85,B 0,C 180,E1 -3553.797,E2 -3553.797} C_VEL
LIN {X 0,Y 547.138,Z 488.704,A -85,B 0,C 180,E1 -3554.818,E2 -3554.818} C_VEL
LIN {X 0,Y 547.636,Z 473.737,A -85,B 0,C 180,E1 -3555.752,E2 -3555.752} C_VEL
LIN {X 0,Y 548.13,Z 458.21,A -85,B 0,C 180,E1 -3556.544,E2 -3556.544} C_VEL
LIN {X 0,Y 548.557,Z 442.08,A -85,B 0,C 180,E1 -3557.195,E2 -3557.195} C_VEL
LIN {X 0,Y 548.865,Z 426.173,A -85,B 0,C 180,E1 -3557.679,E2 -3557.679} C_VEL
LIN {X 0,Y 549.113,Z 409.314,A -85,B 0,C 180,E1 -3558.034,E2 -3558.034} C_VEL
LIN {X 0,Y 550.2,Z 217.152,A -85,B 0,C 180,E1 -3560.683,E2 -3560.683} C_VEL
LIN {X 0,Y 548.112,Z 206.381,A -85,B 0,C 180,E1 -3560.958,E2 -3560.958} C_VEL
LIN {X 0,Y 548.113,Z 201.625,A -85,B 0,C 180,E1 -3561.457,E2 -3561.457} C_VEL
LIN {X 0,Y 545.045,Z 189.908,A -85,B 0,C 180,E1 -3562.891,E2 -3562.891} C_VEL
LIN {X 0,Y 545.062,Z 189.902,A -85,B 0,C 180,E1 -3565.609,E2 -3565.609} C_VEL
LIN {X 0,Y 545.05,Z 189.902,A -85,B 0,C 180,E1 -3568.321,E2 -3568.321} C_VEL
LIN {X 0,Y 545.057,Z 189.906,A -85,B 0,C 180,E1 -3571.256,E2 -3571.256} C_VEL
LIN {X 0,Y 545.035,Z 189.902,A -85,B 0,C 180,E1 -3573.997,E2 -3573.997} C_VEL
LIN {X 0,Y 545.065,Z 189.9,A -85,B 0,C 180,E1 -3576.44,E2 -3576.44} C_VEL
LIN {X 0,Y 545.083,Z 189.896,A -85,B 0,C 180,E1 -3579.628,E2 -3579.628} C_VEL
LIN {X 0,Y 545.066,Z 189.906,A -85,B 0,C 180,E1 -3582.749,E2 -3582.749} C_VEL
LIN {X 0,Y 545.085,Z 189.895,A -85,B 0,C 180,E1 -3585.82,E2 -3585.82} C_VEL
LIN {X 0,Y 545.109,Z 189.897,A -85,B 0,C 180,E1 -3588.849,E2 -3588.849} C_VEL
LIN {X 0,Y 545.091,Z 189.895,A -85,B 0,C 180,E1 -3591.847,E2 -3591.847} C_VEL
LIN {X 0,Y 545.193,Z 189.885,A -85,B 0,C 180,E1 -3594.823,E2 -3594.823} C_VEL
LIN {X 0,Y 545.184,Z 189.884,A -85,B 0,C 180,E1 -3597.784,E2 -3597.784} C_VEL
LIN {X 0,Y 545.209,Z 189.882,A -85,B 0,C 180,E1 -3600.739,E2 -3600.739} C_VEL
LIN {X 0,Y 545.167,Z 189.884,A -85,B 0,C 180,E1 -3602.956,E2 -3602.956} C_VEL
LIN {X 0,Y 545.162,Z 189.89,A -85,B 0,C 180,E1 -3605.92,E2 -3605.92} C_VEL
LIN {X 0,Y 545.115,Z 189.891,A -85,B 0,C 180,E1 -3608.9,E2 -3608.9} C_VEL
LIN {X 0,Y 545.128,Z 189.896,A -85,B 0,C 180,E1 -3611.904,E2 -3611.904} C_VEL
LIN {X 0,Y 545.079,Z 189.895,A -85,B 0,C 180,E1 -3614.944,E2 -3614.944} C_VEL
LIN {X 0,Y 545.076,Z 189.902,A -85,B 0,C 180,E1 -3618.026,E2 -3618.026} C_VEL
LIN {X 0,Y 545.089,Z 189.896,A -85,B 0,C 180,E1 -3620.372,E2 -3620.372} C_VEL
LIN {X 0,Y 545.085,Z 189.902,A -85,B 0,C 180,E1 -3623.559,E2 -3623.559} C_VEL
LIN {X 0,Y 545.083,Z 189.898,A -85,B 0,C 180,E1 -3626,E2 -3626} C_VEL
LIN {X 0,Y 545.084,Z 189.895,A -85,B 0,C 180,E1 -3628.749,E2 -3628.749} C_VEL
LIN {X 0,Y 545.072,Z 189.904,A -85,B 0,C 180,E1 -3631.683,E2 -3631.683} C_VEL
LIN {X 0,Y 545.073,Z 189.898,A -85,B 0,C 180,E1 -3634.564,E2 -3634.564} C_VEL
LIN {X 0,Y 545.031,Z 189.912,A -85,B 0,C 180,E1 -3637.304,E2 -3637.304} C_VEL
LIN {X 0,Y 545.068,Z 189.899,A -85,B 0,C 180,E1 -3640.142,E2 -3640.142} C_VEL
LIN {X 0,Y 545.074,Z 189.906,A -85,B 0,C 180,E1 -3643.107,E2 -3643.107} C_VEL
LIN {X 0,Y 545.044,Z 189.902,A -85,B 0,C 180,E1 -3646.227,E2 -3646.227} C_VEL
LIN {X 0,Y 545.076,Z 189.905,A -85,B 0,C 180,E1 -3648.886,E2 -3648.886} C_VEL
LIN {X 0,Y 545.078,Z 189.903,A -85,B 0,C 180,E1 -3650.819,E2 -3650.819} C_VEL
LIN {X 0,Y 545.037,Z 189.903,A -85,B 0,C 180,E1 -3653.62,E2 -3653.62} C_VEL
LIN {X 0,Y 545.061,Z 189.9,A -85,B 0,C 180,E1 -3656.329,E2 -3656.329} C_VEL
LIN {X 0,Y 545.061,Z 189.907,A -85,B 0,C 180,E1 -3658.953,E2 -3658.953} C_VEL
LIN {X 0,Y 545.055,Z 189.934,A -85,B 0,C 180,E1 -3660.819,E2 -3660.819} C_VEL
LIN {X 0,Y 548.758,Z 202.51,A -85,B 0,C 180,E1 -3662.199,E2 -3662.199} C_VEL
LIN {X 0,Y 548.761,Z 210.711,A -85,B 0,C 180,E1 -3662.958,E2 -3662.958} C_VEL
LIN {X 0,Y 548.15,Z 234.298,A -85,B 0,C 180,E1 -3665.09,E2 -3665.09} C_VEL
LIN {X 0,Y 550.254,Z 246.392,A -85,B 0,C 180,E1 -3665.371,E2 -3665.371} C_VEL
LIN {X 0,Y 549.05,Z 440.422,A -85,B 0,C 180,E1 -3668.037,E2 -3668.037} C_VEL
LIN {X 0,Y 548.827,Z 456.801,A -85,B 0,C 180,E1 -3668.398,E2 -3668.398} C_VEL
LIN {X 0,Y 548.436,Z 473.665,A -85,B 0,C 180,E1 -3668.924,E2 -3668.924} C_VEL
LIN {X 0,Y 548.055,Z 489.895,A -85,B 0,C 180,E1 -3669.595,E2 -3669.595} C_VEL
LIN {X 0,Y 547.625,Z 503.946,A -85,B 0,C 180,E1 -3670.313,E2 -3670.313} C_VEL
LIN {X 0,Y 547.153,Z 519.271,A -85,B 0,C 180,E1 -3671.27,E2 -3671.27} C_VEL
LIN {X 0,Y 546.629,Z 533.211,A -85,B 0,C 180,E1 -3672.317,E2 -3672.317} C_VEL
LIN {X 0,Y 546.157,Z 547.068,A -85,B 0,C 180,E1 -3673.555,E2 -3673.555} C_VEL
LIN {X 0,Y 545.804,Z 558.335,A -85,B 0,C 180,E1 -3674.733,E2 -3674.733} C_VEL
LIN {X 0,Y 545.467,Z 568.908,A -85,B 0,C 180,E1 -3676.02,E2 -3676.02} C_VEL
LIN {X 0,Y 545.227,Z 578.209,A -85,B 0,C 180,E1 -3677.342,E2 -3677.342} C_VEL
LIN {X 0,Y 545.017,Z 587.269,A -85,B 0,C 180,E1 -3678.848,E2 -3678.848} C_VEL
LIN {X 0,Y 544.795,Z 594.857,A -85,B 0,C 180,E1 -3680.346,E2 -3680.346} C_VEL
LIN {X 0,Y 544.738,Z 602.466,A -85,B 0,C 180,E1 -3682.215,E2 -3682.215} C_VEL
LIN {X 0,Y 544.687,Z 608.25,A -85,B 0,C 180,E1 -3684.076,E2 -3684.076} C_VEL
LIN {X 0,Y 544.599,Z 611.635,A -85,B 0,C 180,E1 -3685.559,E2 -3685.559} C_VEL
LIN {X 0,Y 544.638,Z 614.091,A -85,B 0,C 180,E1 -3687.042,E2 -3687.042} C_VEL
LIN {X 0,Y 544.54,Z 615.479,A -85,B 0,C 180,E1 -3688.521,E2 -3688.521} C_VEL
LIN {X 0,Y 544.536,Z 616,A -85,B 0,C 180,E1 -3690,E2 -3690} C_VEL
LIN {X 0,Y 544.54,Z 615.478,A -85,B 0,C 180,E1 -3691.479,E2 -3691.479} C_VEL
LIN {X 0,Y 544.638,Z 614.089,A -85,B 0,C 180,E1 -3692.959,E2 -3692.959} C_VEL
LIN {X 0,Y 544.6,Z 611.634,A -85,B 0,C 180,E1 -3694.441,E2 -3694.441} C_VEL
LIN {X 0,Y 544.686,Z 608.251,A -85,B 0,C 180,E1 -3695.925,E2 -3695.925} C_VEL
LIN {X 0,Y 544.739,Z 602.467,A -85,B 0,C 180,E1 -3697.786,E2 -3697.786} C_VEL
LIN {X 0,Y 544.795,Z 594.855,A -85,B 0,C 180,E1 -3699.654,E2 -3699.654} C_VEL
LIN {X 0,Y 545.017,Z 587.267,A -85,B 0,C 180,E1 -3701.153,E2 -3701.153} C_VEL
LIN {X 0,Y 545.228,Z 578.207,A -85,B 0,C 180,E1 -3702.658,E2 -3702.658} C_VEL
LIN {X 0,Y 545.53,Z 567.42,A -85,B 0,C 180,E1 -3704.169,E2 -3704.169} C_VEL
LIN {X 0,Y 545.926,Z 556.284,A -85,B 0,C 180,E1 -3705.493,E2 -3705.493} C_VEL
LIN {X 0,Y 546.263,Z 544.137,A -85,B 0,C 180,E1 -3706.73,E2 -3706.73} C_VEL
LIN {X 0,Y 546.72,Z 531.353,A -85,B 0,C 180,E1 -3707.833,E2 -3707.833} C_VEL
LIN {X 0,Y 547.152,Z 517.828,A -85,B 0,C 180,E1 -3708.828,E2 -3708.828} C_VEL
LIN {X 0,Y 547.617,Z 503.941,A -85,B 0,C 180,E1 -3709.687,E2 -3709.687} C_VEL
LIN {X 0,Y 548.124,Z 487.958,A -85,B 0,C 180,E1 -3710.498,E2 -3710.498} C_VEL
LIN {X 0,Y 548.479,Z 472.383,A -85,B 0,C 180,E1 -3711.124,E2 -3711.124} C_VEL
LIN {X 0,Y 548.844,Z 455.917,A -85,B 0,C 180,E1 -3711.626,E2 -3711.626} C_VEL
LIN {X 0,Y 549.043,Z 440.46,A -85,B 0,C 180,E1 -3711.963,E2 -3711.963} C_VEL
LIN {X 0,Y 550.072,Z 275.615,A -85,B 0,C 180,E1 -3714.227,E2 -3714.227} C_VEL
LIN {X 0,Y 550.2,Z 245.396,A -85,B 0,C 180,E1 -3714.647,E2 -3714.647} C_VEL
LIN {X 0,Y 548.196,Z 234.433,A -85,B 0,C 180,E1 -3714.906,E2 -3714.906} C_VEL
LIN {X 0,Y 548.971,Z 204.315,A -85,B 0,C 180,E1 -3717.635,E2 -3717.635} C_VEL
LIN {X 0,Y 548.316,Z 200.871,A -85,B 0,C 180,E1 -3717.99,E2 -3717.99} C_VEL
LIN {X 0,Y 545.069,Z 189.906,A -85,B 0,C 180,E1 -3719.221,E2 -3719.221} C_VEL
LIN {X 0,Y 545.052,Z 189.899,A -85,B 0,C 180,E1 -3721.915,E2 -3721.915} C_VEL
LIN {X 0,Y 545.058,Z 189.901,A -85,B 0,C 180,E1 -3724.565,E2 -3724.565} C_VEL
LIN {X 0,Y 545.028,Z 189.908,A -85,B 0,C 180,E1 -3727.304,E2 -3727.304} C_VEL
LIN {X 0,Y 545.063,Z 189.896,A -85,B 0,C 180,E1 -3730.143,E2 -3730.143} C_VEL
LIN {X 0,Y 545.042,Z 189.907,A -85,B 0,C 180,E1 -3733.11,E2 -3733.11} C_VEL
LIN {X 0,Y 545.042,Z 189.898,A -85,B 0,C 180,E1 -3736.227,E2 -3736.227} C_VEL
LIN {X 0,Y 545.077,Z 189.902,A -85,B 0,C 180,E1 -3738.885,E2 -3738.885} C_VEL
LIN {X 0,Y 545.044,Z 189.9,A -85,B 0,C 180,E1 -3741.864,E2 -3741.864} C_VEL
LIN {X 0,Y 545.032,Z 189.902,A -85,B 0,C 180,E1 -3744.531,E2 -3744.531} C_VEL
LIN {X 0,Y 545.062,Z 189.898,A -85,B 0,C 180,E1 -3747.211,E2 -3747.211} C_VEL
LIN {X 0,Y 545.057,Z 189.897,A -85,B 0,C 180,E1 -3749.81,E2 -3749.81} C_VEL
LIN {X 0,Y 545.083,Z 189.898,A -85,B 0,C 180,E1 -3752.828,E2 -3752.828} C_VEL
LIN {X 0,Y 545.044,Z 189.898,A -85,B 0,C 180,E1 -3755.631,E2 -3755.631} C_VEL
LIN {X 0,Y 545.061,Z 189.9,A -85,B 0,C 180,E1 -3758.837,E2 -3758.837} C_VEL
LIN {X 0,Y 545.053,Z 189.895,A -85,B 0,C 180,E1 -3761.195,E2 -3761.195} C_VEL
LIN {X 0,Y 545.06,Z 189.897,A -85,B 0,C 180,E1 -3763.521,E2 -3763.521} C_VEL
LIN {X 0,Y 545.089,Z 189.894,A -85,B 0,C 180,E1 -3765.82,E2 -3765.82} C_VEL
LIN {X 0,Y 545.113,Z 189.889,A -85,B 0,C 180,E1 -3768.849,E2 -3768.849} C_VEL
LIN {X 0,Y 545.095,Z 189.894,A -85,B 0,C 180,E1 -3771.847,E2 -3771.847} C_VEL
LIN {X 0,Y 545.196,Z 189.879,A -85,B 0,C 180,E1 -3774.823,E2 -3774.823} C_VEL
LIN {X 0,Y 545.186,Z 189.874,A -85,B 0,C 180,E1 -3777.784,E2 -3777.784} C_VEL
LIN {X 0,Y 545.211,Z 189.881,A -85,B 0,C 180,E1 -3780.739,E2 -3780.739} C_VEL
LIN {X 0,Y 545.168,Z 189.883,A -85,B 0,C 180,E1 -3782.956,E2 -3782.956} C_VEL
LIN {X 0,Y 545.164,Z 189.884,A -85,B 0,C 180,E1 -3785.92,E2 -3785.92} C_VEL
LIN {X 0,Y 545.107,Z 189.892,A -85,B 0,C 180,E1 -3788.9,E2 -3788.9} C_VEL
LIN {X 0,Y 545.132,Z 189.892,A -85,B 0,C 180,E1 -3791.904,E2 -3791.904} C_VEL
LIN {X 0,Y 545.082,Z 189.894,A -85,B 0,C 180,E1 -3794.944,E2 -3794.944} C_VEL
LIN {X 0,Y 545.079,Z 189.898,A -85,B 0,C 180,E1 -3798.026,E2 -3798.026} C_VEL
LIN {X 0,Y 545.092,Z 189.896,A -85,B 0,C 180,E1 -3800.372,E2 -3800.372} C_VEL
LIN {X 0,Y 545.089,Z 189.898,A -85,B 0,C 180,E1 -3803.559,E2 -3803.559} C_VEL
LIN {X 0,Y 545.077,Z 189.9,A -85,B 0,C 180,E1 -3806.001,E2 -3806.001} C_VEL
LIN {X 0,Y 545.09,Z 189.894,A -85,B 0,C 180,E1 -3808.749,E2 -3808.749} C_VEL
LIN {X 0,Y 545.066,Z 189.896,A -85,B 0,C 180,E1 -3811.048,E2 -3811.048} C_VEL
LIN {X 0,Y 545.065,Z 189.901,A -85,B 0,C 180,E1 -3813.796,E2 -3813.796} C_VEL
LIN {X 0,Y 545.072,Z 189.895,A -85,B 0,C 180,E1 -3816.927,E2 -3816.927} C_VEL
LIN {X 0,Y 545.062,Z 189.897,A -85,B 0,C 180,E1 -3817.011,E2 -3817.011} C_VEL
LIN {X 0,Y 544.353,Z 189.991,A -85,B 0,C 180,E1 -3817.628,E2 -3817.628} C_VEL
LIN {X 0,Y 541.487,Z 190.35,A -85,B 0,C 180,E1 -3818.629,E2 -3818.629} C_VEL
LIN {X 0,Y 539.099,Z 190.646,A -85,B 0,C 180,E1 -3819.434,E2 -3819.434} C_VEL
LIN {X 0,Y 538.09,Z 190.769,A -85,B 0,C 180,E1 -3820.056,E2 -3820.056} C_VEL
LIN {X 0,Y 538.015,Z 190.776,A -85,B 0,C 180,E1 -3820.267,E2 -3820.267} C_VEL
LIN {X 0,Y 538.024,Z 190.775,A -85,B 0,C 180,E1 -3822.988,E2 -3822.988} C_VEL
LIN {X 0,Y 538.018,Z 190.776,A -85,B 0,C 180,E1 -3826.186,E2 -3826.186} C_VEL
LIN {X 0,Y 538.046,Z 190.775,A -85,B 0,C 180,E1 -3829.253,E2 -3829.253} C_VEL
LIN {X 0,Y 537.99,Z 190.779,A -85,B 0,C 180,E1 -3832.122,E2 -3832.122} C_VEL
LIN {X 0,Y 538.002,Z 190.777,A -85,B 0,C 180,E1 -3834.916,E2 -3834.916} C_VEL
LIN {X 0,Y 538.025,Z 190.776,A -85,B 0,C 180,E1 -3837.618,E2 -3837.618} C_VEL
LIN {X 0,Y 538.017,Z 190.775,A -85,B 0,C 180,E1 -3840.239,E2 -3840.239} C_VEL
LIN {X 0,Y 538.056,Z 190.772,A -85,B 0,C 180,E1 -3842.796,E2 -3842.796} C_VEL
LIN {X 0,Y 538.048,Z 190.777,A -85,B 0,C 180,E1 -3845.293,E2 -3845.293} C_VEL
LIN {X 0,Y 538.021,Z 190.777,A -85,B 0,C 180,E1 -3848.546,E2 -3848.546} C_VEL
LIN {X 0,Y 538.032,Z 190.772,A -85,B 0,C 180,E1 -3850.94,E2 -3850.94} C_VEL
LIN {X 0,Y 538.017,Z 190.782,A -85,B 0,C 180,E1 -3853.299,E2 -3853.299} C_VEL
LIN {X 0,Y 538.064,Z 190.764,A -85,B 0,C 180,E1 -3855.631,E2 -3855.631} C_VEL
LIN {X 0,Y 538.077,Z 190.774,A -85,B 0,C 180,E1 -3858.701,E2 -3858.701} C_VEL
LIN {X 0,Y 538.085,Z 190.769,A -85,B 0,C 180,E1 -3861.739,E2 -3861.739} C_VEL
LIN {X 0,Y 538.16,Z 190.764,A -85,B 0,C 180,E1 -3864.755,E2 -3864.755} C_VEL
LIN {X 0,Y 538.168,Z 190.76,A -85,B 0,C 180,E1 -3867.755,E2 -3867.755} C_VEL
LIN {X 0,Y 538.129,Z 190.834,A -85,B 0,C 180,E1 -3868.947,E2 -3868.947} C_VEL
LIN {X 0,Y 541.163,Z 202.116,A -85,B 0,C 180,E1 -3870.331,E2 -3870.331} C_VEL
LIN {X 0,Y 541.439,Z 205.869,A -85,B 0,C 180,E1 -3870.744,E2 -3870.744} C_VEL
LIN {X 0,Y 541.451,Z 206.937,A -85,B 0,C 180,E1 -3870.831,E2 -3870.831} C_VEL
LIN {X 0,Y 543.78,Z 218.336,A -85,B 0,C 180,E1 -3871.112,E2 -3871.112} C_VEL
LIN {X 0,Y 542.507,Z 412.248,A -85,B 0,C 180,E1 -3873.827,E2 -3873.827} C_VEL
LIN {X 0,Y 542.248,Z 428.715,A -85,B 0,C 180,E1 -3874.204,E2 -3874.204} C_VEL
LIN {X 0,Y 541.82,Z 444.188,A -85,B 0,C 180,E1 -3874.696,E2 -3874.696} C_VEL
LIN {X 0,Y 541.419,Z 458.892,A -85,B 0,C 180,E1 -3875.306,E2 -3875.306} C_VEL
LIN {X 0,Y 540.953,Z 473.43,A -85,B 0,C 180,E1 -3876.059,E2 -3876.059} C_VEL
LIN {X 0,Y 540.408,Z 488.473,A -85,B 0,C 180,E1 -3877.003,E2 -3877.003} C_VEL
LIN {X 0,Y 539.904,Z 502.556,A -85,B 0,C 180,E1 -3878.065,E2 -3878.065} C_VEL
LIN {X 0,Y 539.384,Z 515.168,A -85,B 0,C 180,E1 -3879.184,E2 -3879.184} C_VEL
LIN {X 0,Y 538.887,Z 527.893,A -85,B 0,C 180,E1 -3880.52,E2 -3880.52} C_VEL
LIN {X 0,Y 538.486,Z 540.203,A -85,B 0,C 180,E1 -3882.053,E2 -3882.053} C_VEL
LIN {X 0,Y 538.128,Z 550.619,A -85,B 0,C 180,E1 -3883.596,E2 -3883.596} C_VEL
LIN {X 0,Y 537.922,Z 559.393,A -85,B 0,C 180,E1 -3885.147,E2 -3885.147} C_VEL
LIN {X 0,Y 537.729,Z 566.782,A -85,B 0,C 180,E1 -3886.71,E2 -3886.71} C_VEL
LIN {X 0,Y 537.645,Z 572.905,A -85,B 0,C 180,E1 -3888.283,E2 -3888.283} C_VEL
LIN {X 0,Y 537.569,Z 577.767,A -85,B 0,C 180,E1 -3889.871,E2 -3889.871} C_VEL
LIN {X 0,Y 537.476,Z 581.501,A -85,B 0,C 180,E1 -3891.476,E2 -3891.476} C_VEL
LIN {X 0,Y 537.436,Z 584.153,A -85,B 0,C 180,E1 -3893.098,E2 -3893.098} C_VEL
LIN {X 0,Y 537.411,Z 585.599,A -85,B 0,C 180,E1 -3894.738,E2 -3894.738} C_VEL
LIN {X 0,Y 537.437,Z 585.932,A -85,B 0,C 180,E1 -3896.398,E2 -3896.398} C_VEL
LIN {X 0,Y 537.439,Z 585.114,A -85,B 0,C 180,E1 -3898.083,E2 -3898.083} C_VEL
LIN {X 0,Y 537.467,Z 582.98,A -85,B 0,C 180,E1 -3899.794,E2 -3899.794} C_VEL
LIN {X 0,Y 537.553,Z 579.504,A -85,B 0,C 180,E1 -3901.53,E2 -3901.53} C_VEL
LIN {X 0,Y 537.582,Z 574.548,A -85,B 0,C 180,E1 -3903.303,E2 -3903.303} C_VEL
LIN {X 0,Y 537.693,Z 569.187,A -85,B 0,C 180,E1 -3904.808,E2 -3904.808} C_VEL
LIN {X 0,Y 537.822,Z 561.754,A -85,B 0,C 180,E1 -3906.481,E2 -3906.481} C_VEL
LIN {X 0,Y 538.032,Z 554.301,A -85,B 0,C 180,E1 -3907.874,E2 -3907.874} C_VEL
LIN {X 0,Y 538.267,Z 545.477,A -85,B 0,C 180,E1 -3909.289,E2 -3909.289} C_VEL
LIN {X 0,Y 538.629,Z 534.964,A -85,B 0,C 180,E1 -3910.722,E2 -3910.722} C_VEL
LIN {X 0,Y 539.052,Z 523.207,A -85,B 0,C 180,E1 -3912.086,E2 -3912.086} C_VEL
LIN {X 0,Y 539.571,Z 510.629,A -85,B 0,C 180,E1 -3913.327,E2 -3913.327} C_VEL
LIN {X 0,Y 540.068,Z 497.688,A -85,B 0,C 180,E1 -3914.415,E2 -3914.415} C_VEL
LIN {X 0,Y 540.623,Z 483.655,A -85,B 0,C 180,E1 -3915.413,E2 -3915.413} C_VEL
LIN {X 0,Y 541.135,Z 468.244,A -85,B 0,C 180,E1 -3916.322,E2 -3916.322} C_VEL
LIN {X 0,Y 541.663,Z 452.247,A -85,B 0,C 180,E1 -3917.076,E2 -3917.076} C_VEL
LIN {X 0,Y 542.06,Z 435.745,A -85,B 0,C 180,E1 -3917.682,E2 -3917.682} C_VEL
LIN {X 0,Y 542.429,Z 419.171,A -85,B 0,C 180,E1 -3918.123,E2 -3918.123} C_VEL
LIN {X 0,Y 542.63,Z 400.746,A -85,B 0,C 180,E1 -3918.443,E2 -3918.443} C_VEL
LIN {X 0,Y 543.792,Z 218.761,A -85,B 0,C 180,E1 -3920.973,E2 -3920.973} C_VEL
LIN {X 0,Y 541.447,Z 206.589,A -85,B 0,C 180,E1 -3921.289,E2 -3921.289} C_VEL
LIN {X 0,Y 541.305,Z 202.92,A -85,B 0,C 180,E1 -3921.687,E2 -3921.687} C_VEL
LIN {X 0,Y 538.021,Z 190.783,A -85,B 0,C 180,E1 -3923.184,E2 -3923.184} C_VEL
LIN {X 0,Y 538.002,Z 190.78,A -85,B 0,C 180,E1 -3925.826,E2 -3925.826} C_VEL
LIN {X 0,Y 538,Z 190.782,A -85,B 0,C 180,E1 -3928.498,E2 -3928.498} C_VEL
LIN {X 0,Y 538.011,Z 190.783,A -85,B 0,C 180,E1 -3931.097,E2 -3931.097} C_VEL
LIN {X 0,Y 537.982,Z 190.782,A -85,B 0,C 180,E1 -3933.63,E2 -3933.63} C_VEL
LIN {X 0,Y 537.998,Z 190.779,A -85,B 0,C 180,E1 -3936.122,E2 -3936.122} C_VEL
LIN {X 0,Y 538.029,Z 190.777,A -85,B 0,C 180,E1 -3939.348,E2 -3939.348} C_VEL
LIN {X 0,Y 538.028,Z 190.779,A -85,B 0,C 180,E1 -3942.468,E2 -3942.468} C_VEL
LIN {X 0,Y 538.055,Z 190.771,A -85,B 0,C 180,E1 -3945.63,E2 -3945.63} C_VEL
LIN {X 0,Y 538.069,Z 190.774,A -85,B 0,C 180,E1 -3948.701,E2 -3948.701} C_VEL
LIN {X 0,Y 538.055,Z 190.771,A -85,B 0,C 180,E1 -3951.739,E2 -3951.739} C_VEL
LIN {X 0,Y 538.111,Z 190.765,A -85,B 0,C 180,E1 -3954.003,E2 -3954.003} C_VEL
LIN {X 0,Y 538.131,Z 190.762,A -85,B 0,C 180,E1 -3957.006,E2 -3957.006} C_VEL
LIN {X 0,Y 538.163,Z 190.762,A -85,B 0,C 180,E1 -3960,E2 -3960} C_VEL
LIN {X 0,Y 538.133,Z 190.76,A -85,B 0,C 180,E1 -3962.994,E2 -3962.994} C_VEL
LIN {X 0,Y 538.115,Z 190.769,A -85,B 0,C 180,E1 -3965.997,E2 -3965.997} C_VEL
LIN {X 0,Y 538.065,Z 190.769,A -85,B 0,C 180,E1 -3969.018,E2 -3969.018} C_VEL
LIN {X 0,Y 538.077,Z 190.776,A -85,B 0,C 180,E1 -3972.063,E2 -3972.063} C_VEL
LIN {X 0,Y 538.039,Z 190.773,A -85,B 0,C 180,E1 -3975.144,E2 -3975.144} C_VEL
LIN {X 0,Y 538.028,Z 190.776,A -85,B 0,C 180,E1 -3978.27,E2 -3978.27} C_VEL
LIN {X 0,Y 538.033,Z 190.774,A -85,B 0,C 180,E1 -3980.652,E2 -3980.652} C_VEL
LIN {X 0,Y 538.018,Z 190.781,A -85,B 0,C 180,E1 -3983.888,E2 -3983.888} C_VEL
LIN {X 0,Y 538.044,Z 190.771,A -85,B 0,C 180,E1 -3986.366,E2 -3986.366} C_VEL
LIN {X 0,Y 538.025,Z 190.776,A -85,B 0,C 180,E1 -3988.934,E2 -3988.934} C_VEL
LIN {X 0,Y 538.022,Z 190.779,A -85,B 0,C 180,E1 -3991.891,E2 -3991.891} C_VEL
LIN {X 0,Y 538.021,Z 190.776,A -85,B 0,C 180,E1 -3994.62,E2 -3994.62} C_VEL
LIN {X 0,Y 537.998,Z 190.785,A -85,B 0,C 180,E1 -3997.17,E2 -3997.17} C_VEL
LIN {X 0,Y 538.023,Z 190.779,A -85,B 0,C 180,E1 -3999.797,E2 -3999.797} C_VEL
LIN {X 0,Y 538.014,Z 190.781,A -85,B 0,C 180,E1 -4002.786,E2 -4002.786} C_VEL
LIN {X 0,Y 538.025,Z 190.784,A -85,B 0,C 180,E1 -4005.141,E2 -4005.141} C_VEL
LIN {X 0,Y 538.025,Z 190.777,A -85,B 0,C 180,E1 -4008.227,E2 -4008.227} C_VEL
LIN {X 0,Y 538.009,Z 190.783,A -85,B 0,C 180,E1 -4011.17,E2 -4011.17} C_VEL
LIN {X 0,Y 537.99,Z 190.781,A -85,B 0,C 180,E1 -4014.089,E2 -4014.089} C_VEL
LIN {X 0,Y 538.026,Z 190.78,A -85,B 0,C 180,E1 -4016.728,E2 -4016.728} C_VEL
LIN {X 0,Y 538.011,Z 190.782,A -85,B 0,C 180,E1 -4019.559,E2 -4019.559} C_VEL
LIN {X 0,Y 538.034,Z 190.975,A -85,B 0,C 180,E1 -4020.522,E2 -4020.522} C_VEL
LIN {X 0,Y 542.187,Z 205.015,A -85,B 0,C 180,E1 -4022.089,E2 -4022.089} C_VEL
LIN {X 0,Y 541.549,Z 231.636,A -85,B 0,C 180,E1 -4024.541,E2 -4024.541} C_VEL
LIN {X 0,Y 541.53,Z 234.606,A -85,B 0,C 180,E1 -4024.781,E2 -4024.781} C_VEL
LIN {X 0,Y 543.77,Z 247.542,A -85,B 0,C 180,E1 -4025.077,E2 -4025.077} C_VEL
LIN {X 0,Y 542.449,Z 439.99,A -85,B 0,C 180,E1 -4027.756,E2 -4027.756} C_VEL
LIN {X 0,Y 542.202,Z 456.45,A -85,B 0,C 180,E1 -4028.121,E2 -4028.121} C_VEL
LIN {X 0,Y 541.797,Z 473.35,A -85,B 0,C 180,E1 -4028.653,E2 -4028.653} C_VEL
LIN {X 0,Y 541.385,Z 488.594,A -85,B 0,C 180,E1 -4029.282,E2 -4029.282} C_VEL
LIN {X 0,Y 540.843,Z 503.659,A -85,B 0,C 180,E1 -4030.056,E2 -4030.056} C_VEL
LIN {X 0,Y 540.291,Z 518.999,A -85,B 0,C 180,E1 -4031.023,E2 -4031.023} C_VEL
LIN {X 0,Y 539.806,Z 532.076,A -85,B 0,C 180,E1 -4032.006,E2 -4032.006} C_VEL
LIN {X 0,Y 539.324,Z 545.049,A -85,B 0,C 180,E1 -4033.146,E2 -4033.146} C_VEL
LIN {X 0,Y 538.948,Z 556.287,A -85,B 0,C 180,E1 -4034.301,E2 -4034.301} C_VEL
LIN {X 0,Y 538.586,Z 567.422,A -85,B 0,C 180,E1 -4035.645,E2 -4035.645} C_VEL
LIN {X 0,Y 538.204,Z 578.208,A -85,B 0,C 180,E1 -4037.174,E2 -4037.174} C_VEL
LIN {X 0,Y 537.989,Z 587.269,A -85,B 0,C 180,E1 -4038.7,E2 -4038.7} C_VEL
LIN {X 0,Y 537.739,Z 594.857,A -85,B 0,C 180,E1 -4040.218,E2 -4040.218} C_VEL
LIN {X 0,Y 537.658,Z 602.466,A -85,B 0,C 180,E1 -4042.112,E2 -4042.112} C_VEL
LIN {X 0,Y 537.587,Z 608.25,A -85,B 0,C 180,E1 -4043.997,E2 -4043.997} C_VEL
LIN {X 0,Y 537.5,Z 611.635,A -85,B 0,C 180,E1 -4045.501,E2 -4045.501} C_VEL
LIN {X 0,Y 537.538,Z 614.091,A -85,B 0,C 180,E1 -4047.002,E2 -4047.002} C_VEL
LIN {X 0,Y 537.445,Z 615.478,A -85,B 0,C 180,E1 -4048.502,E2 -4048.502} C_VEL
LIN {X 0,Y 537.437,Z 616,A -85,B 0,C 180,E1 -4050,E2 -4050} C_VEL
LIN {X 0,Y 537.445,Z 615.478,A -85,B 0,C 180,E1 -4051.499,E2 -4051.499} C_VEL
LIN {X 0,Y 537.538,Z 614.089,A -85,B 0,C 180,E1 -4052.998,E2 -4052.998} C_VEL
LIN {X 0,Y 537.5,Z 611.633,A -85,B 0,C 180,E1 -4054.5,E2 -4054.5} C_VEL
LIN {X 0,Y 537.587,Z 608.252,A -85,B 0,C 180,E1 -4056.003,E2 -4056.003} C_VEL
LIN {X 0,Y 537.659,Z 602.467,A -85,B 0,C 180,E1 -4057.889,E2 -4057.889} C_VEL
LIN {X 0,Y 537.739,Z 594.855,A -85,B 0,C 180,E1 -4059.782,E2 -4059.782} C_VEL
LIN {X 0,Y 537.99,Z 587.266,A -85,B 0,C 180,E1 -4061.3,E2 -4061.3} C_VEL
LIN {X 0,Y 538.205,Z 578.206,A -85,B 0,C 180,E1 -4062.826,E2 -4062.826} C_VEL
LIN {X 0,Y 538.586,Z 567.419,A -85,B 0,C 180,E1 -4064.355,E2 -4064.355} C_VEL
LIN {X 0,Y 538.979,Z 556.283,A -85,B 0,C 180,E1 -4065.698,E2 -4065.698} C_VEL
LIN {X 0,Y 539.414,Z 544.068,A -85,B 0,C 180,E1 -4066.949,E2 -4066.949} C_VEL
LIN {X 0,Y 539.963,Z 529.925,A -85,B 0,C 180,E1 -4068.169,E2 -4068.169} C_VEL
LIN {X 0,Y 540.436,Z 516.15,A -85,B 0,C 180,E1 -4069.169,E2 -4069.169} C_VEL
LIN {X 0,Y 540.877,Z 501.91,A -85,B 0,C 180,E1 -4070.042,E2 -4070.042} C_VEL
LIN {X 0,Y 541.395,Z 487.227,A -85,B 0,C 180,E1 -4070.786,E2 -4070.786} C_VEL
LIN {X 0,Y 541.89,Z 470.802,A -85,B 0,C 180,E1 -4071.443,E2 -4071.443} C_VEL
LIN {X 0,Y 542.228,Z 454.688,A -85,B 0,C 180,E1 -4071.928,E2 -4071.928} C_VEL
LIN {X 0,Y 542.486,Z 438.575,A -85,B 0,C 180,E1 -4072.268,E2 -4072.268} C_VEL
LIN {X 0,Y 543.761,Z 246.686,A -85,B 0,C 180,E1 -4074.937,E2 -4074.937} C_VEL
LIN {X 0,Y 541.5,Z 234.025,A -85,B 0,C 180,E1 -4075.255,E2 -4075.255} C_VEL
LIN {X 0,Y 542.335,Z 206.198,A -85,B 0,C 180,E1 -4077.808,E2 -4077.808} C_VEL
LIN {X 0,Y 540.237,Z 198.316,A -85,B 0,C 180,E1 -4078.67,E2 -4078.67} C_VEL
LIN {X 0,Y 538.015,Z 190.784,A -85,B 0,C 180,E1 -4079.532,E2 -4079.532} C_VEL
LIN {X 0,Y 538.015,Z 190.773,A -85,B 0,C 180,E1 -4082.383,E2 -4082.383} C_VEL
LIN {X 0,Y 537.992,Z 190.786,A -85,B 0,C 180,E1 -4085.085,E2 -4085.085} C_VEL
LIN {X 0,Y 537.986,Z 190.781,A -85,B 0,C 180,E1 -4087.878,E2 -4087.878} C_VEL
LIN {X 0,Y 538.019,Z 190.778,A -85,B 0,C 180,E1 -4090.778,E2 -4090.778} C_VEL
LIN {X 0,Y 538.016,Z 190.776,A -85,B 0,C 180,E1 -4094.073,E2 -4094.073} C_VEL
LIN {X 0,Y 537.977,Z 190.788,A -85,B 0,C 180,E1 -4097.018,E2 -4097.018} C_VEL
LIN {X 0,Y 538.045,Z 190.775,A -85,B 0,C 180,E1 -4099.253,E2 -4099.253} C_VEL
LIN {X 0,Y 537.987,Z 190.78,A -85,B 0,C 180,E1 -4102.122,E2 -4102.122} C_VEL
LIN {X 0,Y 537.993,Z 190.785,A -85,B 0,C 180,E1 -4104.915,E2 -4104.915} C_VEL
LIN {X 0,Y 538.014,Z 190.773,A -85,B 0,C 180,E1 -4107.617,E2 -4107.617} C_VEL
LIN {X 0,Y 538.009,Z 190.777,A -85,B 0,C 180,E1 -4110.238,E2 -4110.238} C_VEL
LIN {X 0,Y 538.053,Z 190.774,A -85,B 0,C 180,E1 -4112.796,E2 -4112.796} C_VEL
LIN {X 0,Y 538.019,Z 190.775,A -85,B 0,C 180,E1 -4115.291,E2 -4115.291} C_VEL
LIN {X 0,Y 538.012,Z 190.778,A -85,B 0,C 180,E1 -4118.042,E2 -4118.042} C_VEL
LIN {X 0,Y 538.076,Z 190.767,A -85,B 0,C 180,E1 -4120.148,E2 -4120.148} C_VEL
LIN {X 0,Y 538.008,Z 190.776,A -85,B 0,C 180,E1 -4123.299,E2 -4123.299} C_VEL
LIN {X 0,Y 538.059,Z 190.769,A -85,B 0,C 180,E1 -4125.631,E2 -4125.631} C_VEL
LIN {X 0,Y 538.073,Z 190.768,A -85,B 0,C 180,E1 -4128.702,E2 -4128.702} C_VEL
LIN {X 0,Y 538.059,Z 190.77,A -85,B 0,C 180,E1 -4131.739,E2 -4131.739} C_VEL
LIN {X 0,Y 538.114,Z 190.766,A -85,B 0,C 180,E1 -4134.003,E2 -4134.003} C_VEL
LIN {X 0,Y 538.134,Z 190.751,A -85,B 0,C 180,E1 -4137.006,E2 -4137.006} C_VEL
LIN {X 0,Y 538.167,Z 190.758,A -85,B 0,C 180,E1 -4140,E2 -4140} C_VEL
LIN {X 0,Y 538.135,Z 190.759,A -85,B 0,C 180,E1 -4142.994,E2 -4142.994} C_VEL
LIN {X 0,Y 538.118,Z 190.763,A -85,B 0,C 180,E1 -4145.997,E2 -4145.997} C_VEL
LIN {X 0,Y 538.058,Z 190.769,A -85,B 0,C 180,E1 -4149.018,E2 -4149.018} C_VEL
LIN {X 0,Y 538.08,Z 190.769,A -85,B 0,C 180,E1 -4152.063,E2 -4152.063} C_VEL
LIN {X 0,Y 538.042,Z 190.771,A -85,B 0,C 180,E1 -4155.144,E2 -4155.144} C_VEL
LIN {X 0,Y 538.031,Z 190.772,A -85,B 0,C 180,E1 -4158.27,E2 -4158.27} C_VEL
LIN {X 0,Y 538.036,Z 190.772,A -85,B 0,C 180,E1 -4160.651,E2 -4160.651} C_VEL
LIN {X 0,Y 538.022,Z 190.78,A -85,B 0,C 180,E1 -4163.887,E2 -4163.887} C_VEL
LIN {X 0,Y 538.039,Z 190.772,A -85,B 0,C 180,E1 -4166.367,E2 -4166.367} C_VEL
LIN {X 0,Y 538.035,Z 190.773,A -85,B 0,C 180,E1 -4168.935,E2 -4168.935} C_VEL
LIN {X 0,Y 538.011,Z 190.778,A -85,B 0,C 180,E1 -4171.888,E2 -4171.888} C_VEL
LIN {X 0,Y 538.029,Z 190.773,A -85,B 0,C 180,E1 -4174.621,E2 -4174.621} C_VEL
LIN {X 0,Y 538.005,Z 190.778,A -85,B 0,C 180,E1 -4177.171,E2 -4177.171} C_VEL
LIN {X 0,Y 538.015,Z 190.776,A -85,B 0,C 180,E1 -4180.267,E2 -4180.267} C_VEL
LIN {X 0,Y 537.366,Z 190.858,A -85,B 0,C 180,E1 -4180.892,E2 -4180.892} C_VEL
LIN {X 0,Y 534.513,Z 191.218,A -85,B 0,C 180,E1 -4181.907,E2 -4181.907} C_VEL
LIN {X 0,Y 532.087,Z 191.523,A -85,B 0,C 180,E1 -4182.724,E2 -4182.724} C_VEL
LIN {X 0,Y 531.038,Z 191.65,A -85,B 0,C 180,E1 -4183.355,E2 -4183.355} C_VEL
LIN {X 0,Y 530.949,Z 191.658,A -85,B 0,C 180,E1 -4183.569,E2 -4183.569} C_VEL
LIN {X 0,Y 530.962,Z 191.654,A -85,B 0,C 180,E1 -4186.506,E2 -4186.506} C_VEL
LIN {X 0,Y 530.979,Z 191.657,A -85,B 0,C 180,E1 -4189.567,E2 -4189.567} C_VEL
LIN {X 0,Y 530.965,Z 191.653,A -85,B 0,C 180,E1 -4192.577,E2 -4192.577} C_VEL
LIN {X 0,Y 530.99,Z 191.656,A -85,B 0,C 180,E1 -4195.31,E2 -4195.31} C_VEL
LIN {X 0,Y 530.97,Z 191.651,A -85,B 0,C 180,E1 -4198.032,E2 -4198.032} C_VEL
LIN {X 0,Y 530.988,Z 191.655,A -85,B 0,C 180,E1 -4200.874,E2 -4200.874} C_VEL
LIN {X 0,Y 531.001,Z 191.655,A -85,B 0,C 180,E1 -4203.256,E2 -4203.256} C_VEL
LIN {X 0,Y 530.984,Z 191.649,A -85,B 0,C 180,E1 -4205.961,E2 -4205.961} C_VEL
LIN {X 0,Y 530.998,Z 191.656,A -85,B 0,C 180,E1 -4209.062,E2 -4209.062} C_VEL
LIN {X 0,Y 530.985,Z 191.651,A -85,B 0,C 180,E1 -4211.479,E2 -4211.479} C_VEL
LIN {X 0,Y 530.994,Z 191.655,A -85,B 0,C 180,E1 -4214.65,E2 -4214.65} C_VEL
LIN {X 0,Y 531.04,Z 191.646,A -85,B 0,C 180,E1 -4217.775,E2 -4217.775} C_VEL
LIN {X 0,Y 531.028,Z 191.653,A -85,B 0,C 180,E1 -4220.862,E2 -4220.862} C_VEL
LIN {X 0,Y 531.036,Z 191.645,A -85,B 0,C 180,E1 -4223.159,E2 -4223.159} C_VEL
LIN {X 0,Y 531.119,Z 191.64,A -85,B 0,C 180,E1 -4224.685,E2 -4224.685} C_VEL
LIN {X 0,Y 531.14,Z 191.636,A -85,B 0,C 180,E1 -4227.725,E2 -4227.725} C_VEL
LIN {X 0,Y 531.039,Z 191.652,A -85,B 0,C 180,E1 -4228.625,E2 -4228.625} C_VEL
LIN {X 0,Y 534.413,Z 203.897,A -85,B 0,C 180,E1 -4230.152,E2 -4230.152} C_VEL
LIN {X 0,Y 534.799,Z 207.031,A -85,B 0,C 180,E1 -4230.494,E2 -4230.494} C_VEL
LIN {X 0,Y 537.292,Z 219.105,A -85,B 0,C 180,E1 -4230.799,E2 -4230.799} C_VEL
LIN {X 0,Y 536.304,Z 360.518,A -85,B 0,C 180,E1 -4232.793,E2 -4232.793} C_VEL
LIN {X 0,Y 535.932,Z 413.358,A -85,B 0,C 180,E1 -4233.558,E2 -4233.558} C_VEL
LIN {X 0,Y 535.638,Z 429.763,A -85,B 0,C 180,E1 -4233.948,E2 -4233.948} C_VEL
LIN {X 0,Y 535.168,Z 445.549,A -85,B 0,C 180,E1 -4234.467,E2 -4234.467} C_VEL
LIN {X 0,Y 534.68,Z 462.045,A -85,B 0,C 180,E1 -4235.184,E2 -4235.184} C_VEL
LIN {X 0,Y 534.078,Z 477.771,A -85,B 0,C 180,E1 -4236.043,E2 -4236.043} C_VEL
LIN {X 0,Y 533.584,Z 492.093,A -85,B 0,C 180,E1 -4236.998,E2 -4236.998} C_VEL
LIN {X 0,Y 533.001,Z 504.99,A -85,B 0,C 180,E1 -4238.02,E2 -4238.02} C_VEL
LIN {X 0,Y 532.461,Z 516.846,A -85,B 0,C 180,E1 -4239.113,E2 -4239.113} C_VEL
LIN {X 0,Y 531.928,Z 529.365,A -85,B 0,C 180,E1 -4240.467,E2 -4240.467} C_VEL
LIN {X 0,Y 531.521,Z 540.698,A -85,B 0,C 180,E1 -4241.915,E2 -4241.915} C_VEL
LIN {X 0,Y 531.153,Z 550.424,A -85,B 0,C 180,E1 -4243.388,E2 -4243.388} C_VEL
LIN {X 0,Y 530.891,Z 558.869,A -85,B 0,C 180,E1 -4244.899,E2 -4244.899} C_VEL
LIN {X 0,Y 530.654,Z 566.61,A -85,B 0,C 180,E1 -4246.543,E2 -4246.543} C_VEL
LIN {X 0,Y 530.561,Z 572.766,A -85,B 0,C 180,E1 -4248.136,E2 -4248.136} C_VEL
LIN {X 0,Y 530.475,Z 577.912,A -85,B 0,C 180,E1 -4249.841,E2 -4249.841} C_VEL
LIN {X 0,Y 530.402,Z 580.613,A -85,B 0,C 180,E1 -4250.962,E2 -4250.962} C_VEL
LIN {X 0,Y 530.334,Z 583.498,A -85,B 0,C 180,E1 -4252.6,E2 -4252.6} C_VEL
LIN {X 0,Y 530.309,Z 585.309,A -85,B 0,C 180,E1 -4254.257,E2 -4254.257} C_VEL
LIN {X 0,Y 530.348,Z 585.983,A -85,B 0,C 180,E1 -4255.931,E2 -4255.931} C_VEL
LIN {X 0,Y 530.358,Z 585.436,A -85,B 0,C 180,E1 -4257.632,E2 -4257.632} C_VEL
LIN {X 0,Y 530.376,Z 583.691,A -85,B 0,C 180,E1 -4259.359,E2 -4259.359} C_VEL
LIN {X 0,Y 530.43,Z 580.647,A -85,B 0,C 180,E1 -4261.113,E2 -4261.113} C_VEL
LIN {X 0,Y 530.454,Z 576.105,A -85,B 0,C 180,E1 -4262.902,E2 -4262.902} C_VEL
LIN {X 0,Y 530.577,Z 571.648,A -85,B 0,C 180,E1 -4264.26,E2 -4264.26} C_VEL
LIN {X 0,Y 530.69,Z 565.212,A -85,B 0,C 180,E1 -4265.878,E2 -4265.878} C_VEL
LIN {X 0,Y 530.888,Z 557.222,A -85,B 0,C 180,E1 -4267.513,E2 -4267.513} C_VEL
LIN {X 0,Y 531.15,Z 548.489,A -85,B 0,C 180,E1 -4269.014,E2 -4269.014} C_VEL
LIN {X 0,Y 531.529,Z 539.179,A -85,B 0,C 180,E1 -4270.382,E2 -4270.382} C_VEL
LIN {X 0,Y 531.971,Z 527.462,A -85,B 0,C 180,E1 -4271.848,E2 -4271.848} C_VEL
LIN {X 0,Y 532.581,Z 514.642,A -85,B 0,C 180,E1 -4273.199,E2 -4273.199} C_VEL
LIN {X 0,Y 533.186,Z 500.807,A -85,B 0,C 180,E1 -4274.426,E2 -4274.426} C_VEL
LIN {X 0,Y 533.72,Z 487.259,A -85,B 0,C 180,E1 -4275.436,E2 -4275.436} C_VEL
LIN {X 0,Y 534.281,Z 472.779,A -85,B 0,C 180,E1 -4276.341,E2 -4276.341} C_VEL
LIN {X 0,Y 534.884,Z 457.19,A -85,B 0,C 180,E1 -4277.136,E2 -4277.136} C_VEL
LIN {X 0,Y 535.322,Z 440.994,A -85,B 0,C 180,E1 -4277.792,E2 -4277.792} C_VEL
LIN {X 0,Y 535.746,Z 423.904,A -85,B 0,C 180,E1 -4278.303,E2 -4278.303} C_VEL
LIN {X 0,Y 535.993,Z 407.395,A -85,B 0,C 180,E1 -4278.634,E2 -4278.634} C_VEL
LIN {X 0,Y 537.387,Z 220.666,A -85,B 0,C 180,E1 -4281.266,E2 -4281.266} C_VEL
LIN {X 0,Y 535.599,Z 210.683,A -85,B 0,C 180,E1 -4281.504,E2 -4281.504} C_VEL
LIN {X 0,Y 534.775,Z 206.937,A -85,B 0,C 180,E1 -4281.614,E2 -4281.614} C_VEL
LIN {X 0,Y 534.274,Z 203.612,A -85,B 0,C 180,E1 -4282.001,E2 -4282.001} C_VEL
LIN {X 0,Y 530.963,Z 191.661,A -85,B 0,C 180,E1 -4283.507,E2 -4283.507} C_VEL
LIN {X 0,Y 530.955,Z 191.658,A -85,B 0,C 180,E1 -4286.5,E2 -4286.5} C_VEL
LIN {X 0,Y 530.953,Z 191.663,A -85,B 0,C 180,E1 -4289.357,E2 -4289.357} C_VEL
LIN {X 0,Y 530.957,Z 191.659,A -85,B 0,C 180,E1 -4291.542,E2 -4291.542} C_VEL
LIN {X 0,Y 530.954,Z 191.657,A -85,B 0,C 180,E1 -4294.167,E2 -4294.167} C_VEL
LIN {X 0,Y 530.943,Z 191.662,A -85,B 0,C 180,E1 -4296.603,E2 -4296.603} C_VEL
LIN {X 0,Y 530.99,Z 191.658,A -85,B 0,C 180,E1 -4299.062,E2 -4299.062} C_VEL
LIN {X 0,Y 530.977,Z 191.654,A -85,B 0,C 180,E1 -4301.478,E2 -4301.478} C_VEL
LIN {X 0,Y 530.987,Z 191.655,A -85,B 0,C 180,E1 -4304.65,E2 -4304.65} C_VEL
LIN {X 0,Y 531.032,Z 191.643,A -85,B 0,C 180,E1 -4307.775,E2 -4307.775} C_VEL
LIN {X 0,Y 531.015,Z 191.652,A -85,B 0,C 180,E1 -4310.862,E2 -4310.862} C_VEL
LIN {X 0,Y 531.067,Z 191.642,A -85,B 0,C 180,E1 -4313.923,E2 -4313.923} C_VEL
LIN {X 0,Y 531.098,Z 191.639,A -85,B 0,C 180,E1 -4316.966,E2 -4316.966} C_VEL
LIN {X 0,Y 531.134,Z 191.638,A -85,B 0,C 180,E1 -4320,E2 -4320} C_VEL
LIN {X 0,Y 531.099,Z 191.636,A -85,B 0,C 180,E1 -4323.034,E2 -4323.034} C_VEL
LIN {X 0,Y 531.075,Z 191.646,A -85,B 0,C 180,E1 -4326.077,E2 -4326.077} C_VEL
LIN {X 0,Y 531.025,Z 191.646,A -85,B 0,C 180,E1 -4329.138,E2 -4329.138} C_VEL
LIN {X 0,Y 531.034,Z 191.651,A -85,B 0,C 180,E1 -4332.225,E2 -4332.225} C_VEL
LIN {X 0,Y 530.989,Z 191.653,A -85,B 0,C 180,E1 -4335.35,E2 -4335.35} C_VEL
LIN {X 0,Y 531.01,Z 191.655,A -85,B 0,C 180,E1 -4337.722,E2 -4337.722} C_VEL
LIN {X 0,Y 530.993,Z 191.651,A -85,B 0,C 180,E1 -4340.938,E2 -4340.938} C_VEL
LIN {X 0,Y 530.974,Z 191.654,A -85,B 0,C 180,E1 -4344.225,E2 -4344.225} C_VEL
LIN {X 0,Y 531.006,Z 191.648,A -85,B 0,C 180,E1 -4346.743,E2 -4346.743} C_VEL
LIN {X 0,Y 530.976,Z 191.658,A -85,B 0,C 180,E1 -4349.323,E2 -4349.323} C_VEL
LIN {X 0,Y 530.974,Z 191.655,A -85,B 0,C 180,E1 -4352.103,E2 -4352.103} C_VEL
LIN {X 0,Y 530.976,Z 191.656,A -85,B 0,C 180,E1 -4354.853,E2 -4354.853} C_VEL
LIN {X 0,Y 530.96,Z 191.662,A -85,B 0,C 180,E1 -4357.508,E2 -4357.508} C_VEL
LIN {X 0,Y 530.979,Z 191.654,A -85,B 0,C 180,E1 -4360.433,E2 -4360.433} C_VEL
LIN {X 0,Y 530.958,Z 191.664,A -85,B 0,C 180,E1 -4363.282,E2 -4363.282} C_VEL
LIN {X 0,Y 530.978,Z 191.657,A -85,B 0,C 180,E1 -4365.622,E2 -4365.622} C_VEL
LIN {X 0,Y 530.988,Z 191.656,A -85,B 0,C 180,E1 -4368.565,E2 -4368.565} C_VEL
LIN {X 0,Y 530.953,Z 191.658,A -85,B 0,C 180,E1 -4371.53,E2 -4371.53} C_VEL
LIN {X 0,Y 530.949,Z 191.66,A -85,B 0,C 180,E1 -4374.38,E2 -4374.38} C_VEL
LIN {X 0,Y 530.963,Z 191.661,A -85,B 0,C 180,E1 -4377.134,E2 -4377.134} C_VEL
LIN {X 0,Y 530.993,Z 191.75,A -85,B 0,C 180,E1 -4380.189,E2 -4380.189} C_VEL
LIN {X 0,Y 535.572,Z 207.29,A -85,B 0,C 180,E1 -4381.953,E2 -4381.953} C_VEL
LIN {X 0,Y 534.821,Z 234.161,A -85,B 0,C 180,E1 -4384.439,E2 -4384.439} C_VEL
LIN {X 0,Y 537.323,Z 248.059,A -85,B 0,C 180,E1 -4384.768,E2 -4384.768} C_VEL
LIN {X 0,Y 535.878,Z 439.56,A -85,B 0,C 180,E1 -4387.468,E2 -4387.468} C_VEL
LIN {X 0,Y 535.601,Z 455.179,A -85,B 0,C 180,E1 -4387.812,E2 -4387.812} C_VEL
LIN {X 0,Y 535.204,Z 471.729,A -85,B 0,C 180,E1 -4388.327,E2 -4388.327} C_VEL
LIN {X 0,Y 534.781,Z 486.277,A -85,B 0,C 180,E1 -4388.918,E2 -4388.918} C_VEL
LIN {X 0,Y 534.151,Z 501.597,A -85,B 0,C 180,E1 -4389.695,E2 -4389.695} C_VEL
LIN {X 0,Y 533.639,Z 515.857,A -85,B 0,C 180,E1 -4390.577,E2 -4390.577} C_VEL
LIN {X 0,Y 533.119,Z 529.243,A -85,B 0,C 180,E1 -4391.556,E2 -4391.556} C_VEL
LIN {X 0,Y 532.55,Z 542.775,A -85,B 0,C 180,E1 -4392.727,E2 -4392.727} C_VEL
LIN {X 0,Y 532.075,Z 554.268,A -85,B 0,C 180,E1 -4393.896,E2 -4393.896} C_VEL
LIN {X 0,Y 531.663,Z 566.101,A -85,B 0,C 180,E1 -4395.297,E2 -4395.297} C_VEL
LIN {X 0,Y 531.288,Z 575.703,A -85,B 0,C 180,E1 -4396.615,E2 -4396.615} C_VEL
LIN {X 0,Y 531.019,Z 585.095,A -85,B 0,C 180,E1 -4398.15,E2 -4398.15} C_VEL
LIN {X 0,Y 530.783,Z 593.049,A -85,B 0,C 180,E1 -4399.703,E2 -4399.703} C_VEL
LIN {X 0,Y 530.626,Z 599.625,A -85,B 0,C 180,E1 -4401.239,E2 -4401.239} C_VEL
LIN {X 0,Y 530.56,Z 604.958,A -85,B 0,C 180,E1 -4402.771,E2 -4402.771} C_VEL
LIN {X 0,Y 530.495,Z 608.251,A -85,B 0,C 180,E1 -4403.916,E2 -4403.916} C_VEL
LIN {X 0,Y 530.403,Z 611.634,A -85,B 0,C 180,E1 -4405.44,E2 -4405.44} C_VEL
LIN {X 0,Y 530.444,Z 614.091,A -85,B 0,C 180,E1 -4406.962,E2 -4406.962} C_VEL
LIN {X 0,Y 530.355,Z 615.478,A -85,B 0,C 180,E1 -4408.482,E2 -4408.482} C_VEL
LIN {X 0,Y 530.338,Z 616,A -85,B 0,C 180,E1 -4410,E2 -4410} C_VEL
LIN {X 0,Y 530.355,Z 615.477,A -85,B 0,C 180,E1 -4411.519,E2 -4411.519} C_VEL
LIN {X 0,Y 530.444,Z 614.089,A -85,B 0,C 180,E1 -4413.038,E2 -4413.038} C_VEL
LIN {X 0,Y 530.403,Z 611.633,A -85,B 0,C 180,E1 -4414.56,E2 -4414.56} C_VEL
LIN {X 0,Y 530.495,Z 608.252,A -85,B 0,C 180,E1 -4416.084,E2 -4416.084} C_VEL
LIN {X 0,Y 530.569,Z 602.467,A -85,B 0,C 180,E1 -4417.995,E2 -4417.995} C_VEL
LIN {X 0,Y 530.696,Z 594.855,A -85,B 0,C 180,E1 -4419.913,E2 -4419.913} C_VEL
LIN {X 0,Y 531.001,Z 586.252,A -85,B 0,C 180,E1 -4421.646,E2 -4421.646} C_VEL
LIN {X 0,Y 531.228,Z 576.948,A -85,B 0,C 180,E1 -4423.192,E2 -4423.192} C_VEL
LIN {X 0,Y 531.615,Z 567.311,A -85,B 0,C 180,E1 -4424.547,E2 -4424.547} C_VEL
LIN {X 0,Y 532.033,Z 556.078,A -85,B 0,C 180,E1 -4425.908,E2 -4425.908} C_VEL
LIN {X 0,Y 532.538,Z 543.838,A -85,B 0,C 180,E1 -4427.175,E2 -4427.175} C_VEL
LIN {X 0,Y 533.081,Z 530.578,A -85,B 0,C 180,E1 -4428.337,E2 -4428.337} C_VEL
LIN {X 0,Y 533.578,Z 517.341,A -85,B 0,C 180,E1 -4429.325,E2 -4429.325} C_VEL
LIN {X 0,Y 534.074,Z 503.43,A -85,B 0,C 180,E1 -4430.208,E2 -4430.208} C_VEL
LIN {X 0,Y 534.718,Z 487.447,A -85,B 0,C 180,E1 -4431.035,E2 -4431.035} C_VEL
LIN {X 0,Y 535.207,Z 471.828,A -85,B 0,C 180,E1 -4431.674,E2 -4431.674} C_VEL
LIN {X 0,Y 535.614,Z 456.217,A -85,B 0,C 180,E1 -4432.163,E2 -4432.163} C_VEL
LIN {X 0,Y 535.874,Z 441.217,A -85,B 0,C 180,E1 -4432.507,E2 -4432.507} C_VEL
LIN {X 0,Y 537.022,Z 290.741,A -85,B 0,C 180,E1 -4434.629,E2 -4434.629} C_VEL
LIN {X 0,Y 537.173,Z 246.79,A -85,B 0,C 180,E1 -4435.26,E2 -4435.26} C_VEL
LIN {X 0,Y 534.836,Z 233.916,A -85,B 0,C 180,E1 -4435.584,E2 -4435.584} C_VEL
LIN {X 0,Y 535.606,Z 207.421,A -85,B 0,C 180,E1 -4438.054,E2 -4438.054} C_VEL
LIN {X 0,Y 530.97,Z 191.659,A -85,B 0,C 180,E1 -4439.868,E2 -4439.868} C_VEL
LIN {X 0,Y 530.964,Z 191.65,A -85,B 0,C 180,E1 -4442.867,E2 -4442.867} C_VEL
LIN {X 0,Y 530.947,Z 191.661,A -85,B 0,C 180,E1 -4445.62,E2 -4445.62} C_VEL
LIN {X 0,Y 530.962,Z 191.658,A -85,B 0,C 180,E1 -4448.653,E2 -4448.653} C_VEL
LIN {X 0,Y 530.976,Z 191.657,A -85,B 0,C 180,E1 -4451.437,E2 -4451.437} C_VEL
LIN {X 0,Y 530.969,Z 191.656,A -85,B 0,C 180,E1 -4454.548,E2 -4454.548} C_VEL
LIN {X 0,Y 530.966,Z 191.654,A -85,B 0,C 180,E1 -4457.836,E2 -4457.836} C_VEL
LIN {X 0,Y 530.968,Z 191.655,A -85,B 0,C 180,E1 -4460.555,E2 -4460.555} C_VEL
LIN {X 0,Y 530.951,Z 191.653,A -85,B 0,C 180,E1 -4463.441,E2 -4463.441} C_VEL
LIN {X 0,Y 530.952,Z 191.657,A -85,B 0,C 180,E1 -4466.225,E2 -4466.225} C_VEL
LIN {X 0,Y 530.971,Z 191.653,A -85,B 0,C 180,E1 -4469.355,E2 -4469.355} C_VEL
LIN {X 0,Y 531.008,Z 191.654,A -85,B 0,C 180,E1 -4472.468,E2 -4472.468} C_VEL
LIN {X 0,Y 530.985,Z 191.655,A -85,B 0,C 180,E1 -4474.942,E2 -4474.942} C_VEL
LIN {X 0,Y 530.967,Z 191.657,A -85,B 0,C 180,E1 -4478.247,E2 -4478.247} C_VEL
LIN {X 0,Y 530.98,Z 191.651,A -85,B 0,C 180,E1 -4480.677,E2 -4480.677} C_VEL
LIN {X 0,Y 530.984,Z 191.652,A -85,B 0,C 180,E1 -4483.862,E2 -4483.862} C_VEL
LIN {X 0,Y 530.978,Z 191.656,A -85,B 0,C 180,E1 -4486.217,E2 -4486.217} C_VEL
LIN {X 0,Y 531.032,Z 191.643,A -85,B 0,C 180,E1 -4488.55,E2 -4488.55} C_VEL
LIN {X 0,Y 531.034,Z 191.644,A -85,B 0,C 180,E1 -4491.629,E2 -4491.629} C_VEL
LIN {X 0,Y 531.113,Z 191.634,A -85,B 0,C 180,E1 -4494.685,E2 -4494.685} C_VEL
LIN {X 0,Y 531.131,Z 191.623,A -85,B 0,C 180,E1 -4497.725,E2 -4497.725} C_VEL
LIN {X 0,Y 531.151,Z 191.633,A -85,B 0,C 180,E1 -4500.758,E2 -4500.758} C_VEL
LIN {X 0,Y 531.101,Z 191.635,A -85,B 0,C 180,E1 -4503.034,E2 -4503.034} C_VEL
LIN {X 0,Y 531.078,Z 191.64,A -85,B 0,C 180,E1 -4506.077,E2 -4506.077} C_VEL
LIN {X 0,Y 531.05,Z 191.648,A -85,B 0,C 180,E1 -4508.371,E2 -4508.371} C_VEL
LIN {X 0,Y 531.048,Z 191.642,A -85,B 0,C 180,E1 -4511.672,E2 -4511.672} C_VEL
LIN {X 0,Y 531.028,Z 191.645,A -85,B 0,C 180,E1 -4514.956,E2 -4514.956} C_VEL
LIN {X 0,Y 531.014,Z 191.651,A -85,B 0,C 180,E1 -4517.722,E2 -4517.722} C_VEL
LIN {X 0,Y 530.997,Z 191.648,A -85,B 0,C 180,E1 -4520.938,E2 -4520.938} C_VEL
LIN {X 0,Y 530.977,Z 191.651,A -85,B 0,C 180,E1 -4524.225,E2 -4524.225} C_VEL
LIN {X 0,Y 531.003,Z 191.646,A -85,B 0,C 180,E1 -4526.744,E2 -4526.744} C_VEL
LIN {X 0,Y 530.991,Z 191.653,A -85,B 0,C 180,E1 -4529.322,E2 -4529.322} C_VEL
LIN {X 0,Y 530.967,Z 191.653,A -85,B 0,C 180,E1 -4532.101,E2 -4532.101} C_VEL
LIN {X 0,Y 530.986,Z 191.651,A -85,B 0,C 180,E1 -4534.854,E2 -4534.854} C_VEL
LIN {X 0,Y 530.964,Z 191.659,A -85,B 0,C 180,E1 -4537.508,E2 -4537.508} C_VEL
LIN {X 0,Y 530.979,Z 191.652,A -85,B 0,C 180,E1 -4540.433,E2 -4540.433} C_VEL
LIN {X 0,Y 530.959,Z 191.658,A -85,B 0,C 180,E1 -4543.281,E2 -4543.281} C_VEL
LIN {X 0,Y 530.949,Z 191.658,A -85,B 0,C 180,E1 -4543.569,E2 -4543.569} C_VEL
LIN {X 0,Y 530.278,Z 191.738,A -85,B 0,C 180,E1 -4544.203,E2 -4544.203} C_VEL
LIN {X 0,Y 527.435,Z 192.095,A -85,B 0,C 180,E1 -4545.232,E2 -4545.232} C_VEL
LIN {X 0,Y 525.034,Z 192.395,A -85,B 0,C 180,E1 -4546.06,E2 -4546.06} C_VEL
LIN {X 0,Y 524.002,Z 192.522,A -85,B 0,C 180,E1 -4546.7,E2 -4546.7} C_VEL
LIN {X 0,Y 523.916,Z 192.533,A -85,B 0,C 180,E1 -4546.916,E2 -4546.916} C_VEL
LIN {X 0,Y 523.946,Z 192.53,A -85,B 0,C 180,E1 -4549.921,E2 -4549.921} C_VEL
LIN {X 0,Y 523.905,Z 192.535,A -85,B 0,C 180,E1 -4552.868,E2 -4552.868} C_VEL
LIN {X 0,Y 523.937,Z 192.533,A -85,B 0,C 180,E1 -4555.71,E2 -4555.71} C_VEL
LIN {X 0,Y 523.922,Z 192.528,A -85,B 0,C 180,E1 -4558.456,E2 -4558.456} C_VEL
LIN {X 0,Y 523.938,Z 192.537,A -85,B 0,C 180,E1 -4561.125,E2 -4561.125} C_VEL
LIN {X 0,Y 523.983,Z 192.524,A -85,B 0,C 180,E1 -4563.98,E2 -4563.98} C_VEL
LIN {X 0,Y 523.925,Z 192.528,A -85,B 0,C 180,E1 -4566.27,E2 -4566.27} C_VEL
LIN {X 0,Y 523.945,Z 192.533,A -85,B 0,C 180,E1 -4568.767,E2 -4568.767} C_VEL
LIN {X 0,Y 523.947,Z 192.525,A -85,B 0,C 180,E1 -4571.221,E2 -4571.221} C_VEL
LIN {X 0,Y 523.93,Z 192.533,A -85,B 0,C 180,E1 -4573.639,E2 -4573.639} C_VEL
LIN {X 0,Y 523.939,Z 192.522,A -85,B 0,C 180,E1 -4576.028,E2 -4576.028} C_VEL
LIN {X 0,Y 524.012,Z 192.523,A -85,B 0,C 180,E1 -4578.394,E2 -4578.394} C_VEL
LIN {X 0,Y 524.003,Z 192.525,A -85,B 0,C 180,E1 -4581.516,E2 -4581.516} C_VEL
LIN {X 0,Y 524.08,Z 192.515,A -85,B 0,C 180,E1 -4584.613,E2 -4584.613} C_VEL
LIN {X 0,Y 524.112,Z 192.512,A -85,B 0,C 180,E1 -4587.694,E2 -4587.694} C_VEL
LIN {X 0,Y 524.022,Z 192.668,A -85,B 0,C 180,E1 -4588.319,E2 -4588.319} C_VEL
LIN {X 0,Y 527.898,Z 206.675,A -85,B 0,C 180,E1 -4590.091,E2 -4590.091} C_VEL
LIN {X 0,Y 528.253,Z 207.887,A -85,B 0,C 180,E1 -4590.164,E2 -4590.164} C_VEL
LIN {X 0,Y 530.95,Z 220.762,A -85,B 0,C 180,E1 -4590.497,E2 -4590.497} C_VEL
LIN {X 0,Y 529.393,Z 413.046,A -85,B 0,C 180,E1 -4593.259,E2 -4593.259} C_VEL
LIN {X 0,Y 529.072,Z 429.486,A -85,B 0,C 180,E1 -4593.648,E2 -4593.648} C_VEL
LIN {X 0,Y 528.528,Z 446.503,A -85,B 0,C 180,E1 -4594.216,E2 -4594.216} C_VEL
LIN {X 0,Y 528.057,Z 461.321,A -85,B 0,C 180,E1 -4594.867,E2 -4594.867} C_VEL
LIN {X 0,Y 527.496,Z 475.616,A -85,B 0,C 180,E1 -4595.639,E2 -4595.639} C_VEL
LIN {X 0,Y 526.861,Z 490.339,A -85,B 0,C 180,E1 -4596.606,E2 -4596.606} C_VEL
LIN {X 0,Y 526.263,Z 503.933,A -85,B 0,C 180,E1 -4597.674,E2 -4597.674} C_VEL
LIN {X 0,Y 525.592,Z 517.285,A -85,B 0,C 180,E1 -4598.913,E2 -4598.913} C_VEL
LIN {X 0,Y 525.02,Z 529.207,A -85,B 0,C 180,E1 -4600.216,E2 -4600.216} C_VEL
LIN {X 0,Y 524.573,Z 539.928,A -85,B 0,C 180,E1 -4601.593,E2 -4601.593} C_VEL
LIN {X 0,Y 524.184,Z 550.351,A -85,B 0,C 180,E1 -4603.175,E2 -4603.175} C_VEL
LIN {X 0,Y 523.844,Z 559.162,A -85,B 0,C 180,E1 -4604.768,E2 -4604.768} C_VEL
LIN {X 0,Y 523.595,Z 566.566,A -85,B 0,C 180,E1 -4606.372,E2 -4606.372} C_VEL
LIN {X 0,Y 523.478,Z 572.691,A -85,B 0,C 180,E1 -4607.986,E2 -4607.986} C_VEL
LIN {X 0,Y 523.39,Z 578.472,A -85,B 0,C 180,E1 -4609.958,E2 -4609.958} C_VEL
LIN {X 0,Y 523.264,Z 582.796,A -85,B 0,C 180,E1 -4612.068,E2 -4612.068} C_VEL
LIN {X 0,Y 523.235,Z 584.92,A -85,B 0,C 180,E1 -4613.762,E2 -4613.762} C_VEL
LIN {X 0,Y 523.254,Z 585.885,A -85,B 0,C 180,E1 -4615.454,E2 -4615.454} C_VEL
LIN {X 0,Y 523.273,Z 585.733,A -85,B 0,C 180,E1 -4617.17,E2 -4617.17} C_VEL
LIN {X 0,Y 523.275,Z 584.318,A -85,B 0,C 180,E1 -4618.914,E2 -4618.914} C_VEL
LIN {X 0,Y 523.312,Z 581.499,A -85,B 0,C 180,E1 -4620.739,E2 -4620.739} C_VEL
LIN {X 0,Y 523.397,Z 577.518,A -85,B 0,C 180,E1 -4622.486,E2 -4622.486} C_VEL
LIN {X 0,Y 523.501,Z 571.911,A -85,B 0,C 180,E1 -4624.322,E2 -4624.322} C_VEL
LIN {X 0,Y 523.627,Z 565.594,A -85,B 0,C 180,E1 -4625.958,E2 -4625.958} C_VEL
LIN {X 0,Y 523.87,Z 557.403,A -85,B 0,C 180,E1 -4627.673,E2 -4627.673} C_VEL
LIN {X 0,Y 524.21,Z 547.973,A -85,B 0,C 180,E1 -4629.306,E2 -4629.306} C_VEL
LIN {X 0,Y 524.657,Z 537.759,A -85,B 0,C 180,E1 -4630.793,E2 -4630.793} C_VEL
LIN {X 0,Y 525.168,Z 526.17,A -85,B 0,C 180,E1 -4632.227,E2 -4632.227} C_VEL
LIN {X 0,Y 525.773,Z 514.054,A -85,B 0,C 180,E1 -4633.503,E2 -4633.503} C_VEL
LIN {X 0,Y 526.416,Z 500.134,A -85,B 0,C 180,E1 -4634.742,E2 -4634.742} C_VEL
LIN {X 0,Y 527.074,Z 486.141,A -85,B 0,C 180,E1 -4635.782,E2 -4635.782} C_VEL
LIN {X 0,Y 527.696,Z 471.117,A -85,B 0,C 180,E1 -4636.712,E2 -4636.712} C_VEL
LIN {X 0,Y 528.269,Z 456.636,A -85,B 0,C 180,E1 -4637.446,E2 -4637.446} C_VEL
LIN {X 0,Y 528.728,Z 440.364,A -85,B 0,C 180,E1 -4638.104,E2 -4638.104} C_VEL
LIN {X 0,Y 529.18,Z 423.6,A -85,B 0,C 180,E1 -4638.604,E2 -4638.604} C_VEL
LIN {X 0,Y 529.486,Z 405.95,A -85,B 0,C 180,E1 -4638.952,E2 -4638.952} C_VEL
LIN {X 0,Y 530.953,Z 220.84,A -85,B 0,C 180,E1 -4641.594,E2 -4641.594} C_VEL
LIN {X 0,Y 528.128,Z 207.621,A -85,B 0,C 180,E1 -4641.94,E2 -4641.94} C_VEL
LIN {X 0,Y 523.929,Z 192.536,A -85,B 0,C 180,E1 -4643.843,E2 -4643.843} C_VEL
LIN {X 0,Y 523.906,Z 192.537,A -85,B 0,C 180,E1 -4646.633,E2 -4646.633} C_VEL
LIN {X 0,Y 523.936,Z 192.537,A -85,B 0,C 180,E1 -4649.355,E2 -4649.355} C_VEL
LIN {X 0,Y 523.933,Z 192.533,A -85,B 0,C 180,E1 -4652.289,E2 -4652.289} C_VEL
LIN {X 0,Y 523.897,Z 192.538,A -85,B 0,C 180,E1 -4655.427,E2 -4655.427} C_VEL
LIN {X 0,Y 523.93,Z 192.528,A -85,B 0,C 180,E1 -4657.939,E2 -4657.939} C_VEL
LIN {X 0,Y 523.966,Z 192.531,A -85,B 0,C 180,E1 -4660.408,E2 -4660.408} C_VEL
LIN {X 0,Y 523.946,Z 192.535,A -85,B 0,C 180,E1 -4662.837,E2 -4662.837} C_VEL
LIN {X 0,Y 523.969,Z 192.528,A -85,B 0,C 180,E1 -4665.236,E2 -4665.236} C_VEL
LIN {X 0,Y 524.005,Z 192.522,A -85,B 0,C 180,E1 -4668.394,E2 -4668.394} C_VEL
LIN {X 0,Y 523.982,Z 192.523,A -85,B 0,C 180,E1 -4671.516,E2 -4671.516} C_VEL
LIN {X 0,Y 524.029,Z 192.518,A -85,B 0,C 180,E1 -4673.841,E2 -4673.841} C_VEL
LIN {X 0,Y 524.065,Z 192.516,A -85,B 0,C 180,E1 -4676.925,E2 -4676.925} C_VEL
LIN {X 0,Y 524.105,Z 192.513,A -85,B 0,C 180,E1 -4680,E2 -4680} C_VEL
LIN {X 0,Y 524.066,Z 192.512,A -85,B 0,C 180,E1 -4683.075,E2 -4683.075} C_VEL
LIN {X 0,Y 524.038,Z 192.523,A -85,B 0,C 180,E1 -4686.159,E2 -4686.159} C_VEL
LIN {X 0,Y 523.993,Z 192.522,A -85,B 0,C 180,E1 -4689.262,E2 -4689.262} C_VEL
LIN {X 0,Y 523.996,Z 192.525,A -85,B 0,C 180,E1 -4691.74,E2 -4691.74} C_VEL
LIN {X 0,Y 523.986,Z 192.524,A -85,B 0,C 180,E1 -4695.052,E2 -4695.052} C_VEL
LIN {X 0,Y 523.958,Z 192.533,A -85,B 0,C 180,E1 -4697.969,E2 -4697.969} C_VEL
LIN {X 0,Y 523.965,Z 192.527,A -85,B 0,C 180,E1 -4700.41,E2 -4700.41} C_VEL
LIN {X 0,Y 523.91,Z 192.533,A -85,B 0,C 180,E1 -4702.893,E2 -4702.893} C_VEL
LIN {X 0,Y 523.949,Z 192.533,A -85,B 0,C 180,E1 -4705.419,E2 -4705.419} C_VEL
LIN {X 0,Y 523.965,Z 192.529,A -85,B 0,C 180,E1 -4707.999,E2 -4707.999} C_VEL
LIN {X 0,Y 523.941,Z 192.531,A -85,B 0,C 180,E1 -4710.856,E2 -4710.856} C_VEL
LIN {X 0,Y 523.956,Z 192.533,A -85,B 0,C 180,E1 -4713.735,E2 -4713.735} C_VEL
LIN {X 0,Y 523.898,Z 192.536,A -85,B 0,C 180,E1 -4716.402,E2 -4716.402} C_VEL
LIN {X 0,Y 523.917,Z 192.539,A -85,B 0,C 180,E1 -4719.085,E2 -4719.085} C_VEL
LIN {X 0,Y 523.948,Z 192.531,A -85,B 0,C 180,E1 -4722.119,E2 -4722.119} C_VEL
LIN {X 0,Y 523.948,Z 192.536,A -85,B 0,C 180,E1 -4725.309,E2 -4725.309} C_VEL
LIN {X 0,Y 523.951,Z 192.534,A -85,B 0,C 180,E1 -4728.69,E2 -4728.69} C_VEL
LIN {X 0,Y 523.914,Z 192.54,A -85,B 0,C 180,E1 -4731.081,E2 -4731.081} C_VEL
LIN {X 0,Y 523.895,Z 192.537,A -85,B 0,C 180,E1 -4733.826,E2 -4733.826} C_VEL
LIN {X 0,Y 523.937,Z 192.534,A -85,B 0,C 180,E1 -4736.636,E2 -4736.636} C_VEL
LIN {X 0,Y 523.952,Z 192.655,A -85,B 0,C 180,E1 -4739.857,E2 -4739.857} C_VEL
LIN {X 0,Y 528.774,Z 208.819,A -85,B 0,C 180,E1 -4741.729,E2 -4741.729} C_VEL
LIN {X 0,Y 528.797,Z 214.478,A -85,B 0,C 180,E1 -4742.279,E2 -4742.279} C_VEL
LIN {X 0,Y 528.144,Z 233.694,A -85,B 0,C 180,E1 -4744.087,E2 -4744.087} C_VEL
LIN {X 0,Y 530.882,Z 249.552,A -85,B 0,C 180,E1 -4744.465,E2 -4744.465} C_VEL
LIN {X 0,Y 529.318,Z 439.13,A -85,B 0,C 180,E1 -4747.174,E2 -4747.174} C_VEL
LIN {X 0,Y 528.975,Z 455.745,A -85,B 0,C 180,E1 -4747.545,E2 -4747.545} C_VEL
LIN {X 0,Y 528.528,Z 472.72,A -85,B 0,C 180,E1 -4748.09,E2 -4748.09} C_VEL
LIN {X 0,Y 528.073,Z 487.067,A -85,B 0,C 180,E1 -4748.687,E2 -4748.687} C_VEL
LIN {X 0,Y 527.349,Z 503.087,A -85,B 0,C 180,E1 -4749.523,E2 -4749.523} C_VEL
LIN {X 0,Y 526.796,Z 517.019,A -85,B 0,C 180,E1 -4750.416,E2 -4750.416} C_VEL
LIN {X 0,Y 526.153,Z 531.38,A -85,B 0,C 180,E1 -4751.508,E2 -4751.508} C_VEL
LIN {X 0,Y 525.572,Z 544.543,A -85,B 0,C 180,E1 -4752.691,E2 -4752.691} C_VEL
LIN {X 0,Y 525.076,Z 555.816,A -85,B 0,C 180,E1 -4753.876,E2 -4753.876} C_VEL
LIN {X 0,Y 524.632,Z 567.063,A -85,B 0,C 180,E1 -4755.255,E2 -4755.255} C_VEL
LIN {X 0,Y 524.176,Z 577.957,A -85,B 0,C 180,E1 -4756.825,E2 -4756.825} C_VEL
LIN {X 0,Y 523.934,Z 587.115,A -85,B 0,C 180,E1 -4758.393,E2 -4758.393} C_VEL
LIN {X 0,Y 523.658,Z 594.781,A -85,B 0,C 180,E1 -4759.952,E2 -4759.952} C_VEL
LIN {X 0,Y 523.503,Z 602.465,A -85,B 0,C 180,E1 -4761.897,E2 -4761.897} C_VEL
LIN {X 0,Y 523.411,Z 608.251,A -85,B 0,C 180,E1 -4763.834,E2 -4763.834} C_VEL
LIN {X 0,Y 523.312,Z 611.633,A -85,B 0,C 180,E1 -4765.378,E2 -4765.378} C_VEL
LIN {X 0,Y 523.353,Z 614.091,A -85,B 0,C 180,E1 -4766.921,E2 -4766.921} C_VEL
LIN {X 0,Y 523.269,Z 615.478,A -85,B 0,C 180,E1 -4768.461,E2 -4768.461} C_VEL
LIN {X 0,Y 523.242,Z 616,A -85,B 0,C 180,E1 -4770,E2 -4770} C_VEL
LIN {X 0,Y 523.269,Z 615.477,A -85,B 0,C 180,E1 -4771.539,E2 -4771.539} C_VEL
LIN {X 0,Y 523.353,Z 614.089,A -85,B 0,C 180,E1 -4773.079,E2 -4773.079} C_VEL
LIN {X 0,Y 523.312,Z 611.632,A -85,B 0,C 180,E1 -4774.622,E2 -4774.622} C_VEL
LIN {X 0,Y 523.411,Z 608.253,A -85,B 0,C 180,E1 -4776.167,E2 -4776.167} C_VEL
LIN {X 0,Y 523.503,Z 602.467,A -85,B 0,C 180,E1 -4778.104,E2 -4778.104} C_VEL
LIN {X 0,Y 523.658,Z 594.783,A -85,B 0,C 180,E1 -4780.048,E2 -4780.048} C_VEL
LIN {X 0,Y 523.956,Z 586.562,A -85,B 0,C 180,E1 -4781.715,E2 -4781.715} C_VEL
